C07322=1188.641,207.407,-59.713,-177.679,6.703,148.552
C07323=1188.636,207.656,-59.737,-177.676,6.705,148.552
C07324=1188.631,207.905,-59.762,-177.673,6.707,148.552
C07325=1188.627,208.154,-59.786,-177.671,6.709,148.551
C07326=1188.623,208.402,-59.810,-177.668,6.712,148.551
C07327=1188.618,208.651,-59.834,-177.665,6.713,148.551
C07328=1188.613,208.900,-59.858,-177.663,6.715,148.550
C07329=1188.609,209.149,-59.883,-177.660,6.717,148.550
C07330=1188.604,209.398,-59.907,-177.658,6.719,148.550
C07331=1188.599,209.646,-59.932,-177.654,6.722,148.550
C07332=1188.595,209.895,-59.956,-177.652,6.724,148.549
C07333=1188.591,210.144,-59.980,-177.650,6.726,148.549
C07334=1188.586,210.414,-60.007,-177.647,6.728,148.549
C07335=1188.581,210.684,-60.034,-177.644,6.730,148.549
C07336=1188.576,210.955,-60.061,-177.641,6.732,148.548
C07337=1188.571,211.226,-60.087,-177.638,6.735,148.548
C07338=1188.566,211.474,-60.111,-177.635,6.736,148.548
C07339=1188.561,211.722,-60.136,-177.633,6.738,148.547
C07340=1188.558,211.972,-60.161,-177.630,6.741,148.547
C07341=1188.552,212.220,-60.186,-177.627,6.743,148.547
C07342=1188.548,212.469,-60.210,-177.624,6.745,148.547
C07343=1188.543,212.718,-60.235,-177.622,6.747,148.546
C07344=1188.539,212.967,-60.259,-177.619,6.750,148.546
C07345=1188.534,213.215,-60.283,-177.616,6.751,148.546
C07346=1188.530,213.464,-60.308,-177.614,6.753,148.545
C07347=1188.525,213.713,-60.332,-177.612,6.755,148.545
C07348=1188.521,213.962,-60.358,-177.609,6.757,148.545
C07349=1188.516,214.210,-60.382,-177.606,6.760,148.545
C07350=1188.511,214.459,-60.407,-177.604,6.762,148.545
C07351=1188.507,214.708,-60.431,-177.601,6.764,148.544
C07352=1188.502,214.957,-60.456,-177.598,6.766,148.544
C07353=1188.498,215.205,-60.481,-177.595,6.768,148.544
C07354=1188.494,215.454,-60.506,-177.593,6.770,148.543
C07355=1188.489,215.703,-60.531,-177.590,6.772,148.543
C07356=1188.485,215.952,-60.555,-177.588,6.774,148.543
C07357=1188.480,216.200,-60.580,-177.585,6.777,148.543
C07358=1188.475,216.449,-60.605,-177.582,6.779,148.542
C07359=1188.471,216.698,-60.630,-177.580,6.781,148.542
C07360=1188.466,216.947,-60.654,-177.577,6.782,148.542
C07361=1188.462,217.195,-60.680,-177.574,6.785,148.542
C07362=1188.457,217.444,-60.704,-177.571,6.787,148.541
C07363=1188.453,217.693,-60.729,-177.569,6.789,148.541
C07364=1188.448,217.941,-60.754,-177.567,6.791,148.541
C07365=1188.444,218.190,-60.779,-177.563,6.794,148.541
C07366=1188.439,218.439,-60.804,-177.561,6.796,148.540
C07367=1188.434,218.687,-60.829,-177.559,6.798,148.540
C07368=1188.430,218.936,-60.853,-177.556,6.800,148.540
C07369=1188.426,219.185,-60.879,-177.553,6.802,148.539
C07370=1188.421,219.434,-60.904,-177.551,6.804,148.539
C07371=1188.417,219.682,-60.929,-177.548,6.806,148.539
C07372=1188.412,219.931,-60.954,-177.545,6.809,148.539
C07373=1188.407,220.180,-60.978,-177.543,6.811,148.539
C07374=1188.403,220.429,-61.004,-177.540,6.813,148.538
C07375=1188.399,220.677,-61.028,-177.537,6.815,148.538
C07376=1188.394,220.926,-61.054,-177.534,6.818,148.538
C07377=1188.389,221.175,-61.079,-177.532,6.819,148.538
C07378=1188.385,221.423,-61.104,-177.529,6.821,148.537
C07379=1188.380,221.672,-61.129,-177.527,6.823,148.537
C07380=1188.376,221.921,-61.154,-177.524,6.826,148.537
C07381=1188.371,222.169,-61.179,-177.521,6.828,148.536
C07382=1188.367,222.418,-61.205,-177.519,6.830,148.536
C07383=1188.362,222.666,-61.230,-177.516,6.833,148.536
C07384=1188.358,222.916,-61.255,-177.513,6.834,148.536
C07385=1188.353,223.164,-61.280,-177.511,6.837,148.536
C07386=1188.349,223.413,-61.305,-177.508,6.838,148.535
C07387=1188.345,223.662,-61.331,-177.506,6.841,148.535
C07388=1188.340,223.910,-61.356,-177.503,6.843,148.535
C07389=1188.336,224.159,-61.381,-177.500,6.845,148.535
C07390=1188.331,224.407,-61.406,-177.497,6.848,148.534
C07391=1188.327,224.656,-61.432,-177.495,6.850,148.534
C07392=1188.321,224.905,-61.457,-177.492,6.852,148.534
C07393=1188.317,225.154,-61.482,-177.489,6.855,148.534
C07394=1188.313,225.403,-61.508,-177.487,6.856,148.533
C07395=1188.309,225.651,-61.532,-177.485,6.859,148.533
C07396=1188.304,225.900,-61.558,-177.482,6.860,148.533
C07397=1188.300,226.148,-61.583,-177.479,6.863,148.533
C07398=1188.295,226.397,-61.609,-177.477,6.865,148.533
C07399=1188.291,226.646,-61.634,-177.474,6.867,148.532
C07400=1188.286,226.894,-61.660,-177.471,6.870,148.532
C07401=1188.282,227.143,-61.685,-177.469,6.872,148.532
C07402=1188.277,227.391,-61.711,-177.466,6.874,148.531
C07403=1188.273,227.640,-61.737,-177.463,6.877,148.531
C07404=1188.268,227.889,-61.762,-177.461,6.878,148.531
C07405=1188.263,228.137,-61.787,-177.458,6.880,148.531
C07406=1188.259,228.386,-61.813,-177.455,6.883,148.531
C07407=1188.255,228.635,-61.838,-177.452,6.885,148.530
C07408=1188.250,228.883,-61.864,-177.450,6.887,148.530
C07409=1188.246,229.132,-61.890,-177.447,6.890,148.530
C07410=1188.241,229.381,-61.915,-177.445,6.892,148.530
C07411=1188.236,229.629,-61.940,-177.442,6.894,148.529
C07412=1188.232,229.878,-61.966,-177.439,6.896,148.529
C07413=1188.228,230.127,-61.991,-177.437,6.899,148.529
C07414=1188.223,230.375,-62.017,-177.434,6.900,148.529
C07415=1188.218,230.624,-62.043,-177.432,6.903,148.529
C07416=1188.214,230.873,-62.069,-177.429,6.905,148.528
C07417=1188.209,231.121,-62.094,-177.427,6.907,148.528
C07418=1188.205,231.370,-62.120,-177.424,6.910,148.528
C07419=1188.201,231.619,-62.146,-177.421,6.912,148.528
C07420=1188.196,231.867,-62.171,-177.419,6.914,148.528
C07421=1188.192,232.116,-62.197,-177.415,6.917,148.527
C07422=1188.187,232.365,-62.223,-177.413,6.919,148.527
C07423=1188.183,232.613,-62.248,-177.411,6.921,148.527
C07424=1188.178,232.862,-62.274,-177.408,6.924,148.527
C07425=1188.173,233.111,-62.300,-177.405,6.925,148.526
C07426=1188.169,233.359,-62.326,-177.403,6.927,148.526
C07427=1188.165,233.608,-62.352,-177.400,6.930,148.526
C07428=1188.160,233.856,-62.378,-177.398,6.932,148.526
C07429=1188.155,234.105,-62.404,-177.395,6.934,148.526
C07430=1188.151,234.354,-62.430,-177.392,6.937,148.526
C07431=1188.147,234.602,-62.456,-177.390,6.939,148.525
C07432=1188.142,234.850,-62.481,-177.386,6.942,148.525
C07433=1188.138,235.099,-62.507,-177.384,6.944,148.525
C07434=1188.133,235.348,-62.533,-177.382,6.946,148.524
C07435=1188.129,235.597,-62.560,-177.379,6.949,148.524
C07436=1188.125,235.845,-62.585,-177.376,6.950,148.524
C07437=1188.120,236.093,-62.611,-177.374,6.952,148.524
C07438=1188.115,236.366,-62.639,-177.371,6.955,148.524
C07439=1188.110,236.637,-62.668,-177.368,6.958,148.524
C07440=1188.106,236.909,-62.696,-177.365,6.961,148.523
C07441=1188.101,237.179,-62.725,-177.362,6.963,148.523
C07442=1188.096,237.429,-62.751,-177.360,6.966,148.523
C07443=1188.091,237.677,-62.777,-177.357,6.967,148.523
C07444=1188.087,237.926,-62.803,-177.355,6.970,148.523
C07445=1188.082,238.175,-62.829,-177.352,6.972,148.522
C07446=1188.078,238.423,-62.855,-177.349,6.974,148.522
C07447=1188.074,238.671,-62.881,-177.346,6.977,148.522
C07448=1188.069,238.920,-62.908,-177.344,6.979,148.522
C07449=1188.065,239.169,-62.933,-177.341,6.981,148.521
C07450=1188.061,239.417,-62.960,-177.339,6.984,148.521
C07451=1188.056,239.666,-62.986,-177.336,6.986,148.521
C07452=1188.051,239.915,-63.012,-177.333,6.989,148.521
C07453=1188.047,240.162,-63.038,-177.331,6.991,148.521
C07454=1188.042,240.412,-63.064,-177.328,6.993,148.521
C07455=1188.038,240.660,-63.091,-177.326,6.996,148.521
C07456=1188.033,240.909,-63.117,-177.323,6.998,148.520
C07457=1188.029,241.157,-63.144,-177.320,7.001,148.520
C07458=1188.025,241.406,-63.169,-177.318,7.002,148.520
C07459=1188.020,241.654,-63.197,-177.316,7.004,148.520
C07460=1188.016,241.903,-63.222,-177.312,7.007,148.519
C07461=1188.011,242.152,-63.249,-177.310,7.009,148.519
C07462=1188.007,242.400,-63.275,-177.307,7.012,148.519
C07463=1188.002,242.648,-63.302,-177.305,7.014,148.519
C07464=1187.998,242.897,-63.328,-177.302,7.016,148.519
C07465=1187.993,243.146,-63.355,-177.299,7.019,148.519
C07466=1187.989,243.394,-63.380,-177.297,7.021,148.518
C07467=1187.984,243.643,-63.407,-177.294,7.024,148.518
C07468=1187.980,243.892,-63.433,-177.292,7.026,148.518
C07469=1187.975,244.140,-63.460,-177.289,7.029,148.518
C07470=1187.971,244.388,-63.487,-177.287,7.031,148.518
C07471=1187.966,244.637,-63.513,-177.284,7.033,148.517
C07472=1187.962,244.886,-63.540,-177.281,7.036,148.517
C07473=1187.958,245.134,-63.567,-177.279,7.038,148.517
C07474=1187.954,245.383,-63.592,-177.276,7.040,148.517
C07475=1187.949,245.631,-63.619,-177.274,7.042,148.517
C07476=1187.945,245.880,-63.646,-177.270,7.045,148.517
C07477=1187.940,246.129,-63.672,-177.268,7.047,148.516
C07478=1187.936,246.377,-63.699,-177.265,7.050,148.516
C07479=1187.931,246.625,-63.726,-177.263,7.052,148.516
C07480=1187.927,246.875,-63.752,-177.261,7.054,148.516
C07481=1187.923,247.123,-63.779,-177.258,7.057,148.516
C07482=1187.918,247.371,-63.806,-177.255,7.059,148.516
C07483=1187.914,247.619,-63.832,-177.252,7.062,148.515
C07484=1187.909,247.869,-63.858,-177.250,7.064,148.515
C07485=1187.904,248.117,-63.885,-177.247,7.067,148.515
C07486=1187.900,248.365,-63.912,-177.245,7.069,148.515
C07487=1187.896,248.614,-63.939,-177.242,7.072,148.515
C07488=1187.891,248.862,-63.966,-177.240,7.074,148.515
C07489=1187.887,249.110,-63.993,-177.237,7.076,148.514
C07490=1187.882,249.359,-64.019,-177.234,7.079,148.514
C07491=1187.878,249.608,-64.046,-177.232,7.080,148.514
C07492=1187.874,249.856,-64.072,-177.229,7.083,148.514
C07493=1187.869,250.105,-64.099,-177.227,7.086,148.514
C07494=1187.864,250.353,-64.127,-177.224,7.088,148.514
C07495=1187.860,250.602,-64.154,-177.221,7.090,148.514
C07496=1187.856,250.851,-64.180,-177.219,7.093,148.513
C07497=1187.852,251.099,-64.207,-177.216,7.095,148.513
C07498=1187.847,251.348,-64.235,-177.213,7.098,148.513
C07499=1187.842,251.596,-64.262,-177.211,7.100,148.513
C07500=1187.839,251.844,-64.288,-177.208,7.103,148.513
C07501=1187.834,252.093,-64.315,-177.206,7.105,148.513
C07502=1187.829,252.341,-64.342,-177.203,7.108,148.512
C07503=1187.825,252.590,-64.369,-177.200,7.110,148.512
C07504=1187.821,252.838,-64.396,-177.198,7.113,148.512
C07505=1187.817,253.087,-64.423,-177.195,7.115,148.512
C07506=1187.812,253.336,-64.450,-177.192,7.118,148.512
C07507=1187.807,253.584,-64.477,-177.190,7.120,148.512
C07508=1187.803,253.833,-64.504,-177.187,7.123,148.511
C07509=1187.799,254.081,-64.531,-177.185,7.125,148.511
C07510=1187.794,254.329,-64.558,-177.182,7.128,148.511
C07511=1187.789,254.578,-64.585,-177.180,7.130,148.511
C07512=1187.785,254.827,-64.612,-177.177,7.133,148.511
C07513=1187.781,255.075,-64.639,-177.175,7.135,148.511
C07514=1187.776,255.323,-64.667,-177.171,7.137,148.511
C07515=1187.772,255.572,-64.694,-177.169,7.140,148.510
C07516=1187.768,255.820,-64.721,-177.167,7.143,148.510
C07517=1187.764,256.069,-64.748,-177.164,7.145,148.510
C07518=1187.759,256.318,-64.775,-177.161,7.147,148.510
C07519=1187.755,256.566,-64.803,-177.159,7.150,148.510
C07520=1187.750,256.814,-64.830,-177.156,7.153,148.510
C07521=1187.745,257.063,-64.857,-177.154,7.154,148.510
C07522=1187.741,257.312,-64.885,-177.151,7.157,148.510
C07523=1187.737,257.560,-64.912,-177.149,7.160,148.509
C07524=1187.732,257.808,-64.939,-177.146,7.162,148.509
C07525=1187.728,258.057,-64.966,-177.143,7.165,148.509
C07526=1187.723,258.305,-64.993,-177.141,7.167,148.509
C07527=1187.719,258.554,-65.022,-177.138,7.170,148.509
C07528=1187.715,258.802,-65.049,-177.135,7.172,148.509
C07529=1187.710,259.051,-65.076,-177.133,7.175,148.509
C07530=1187.706,259.299,-65.104,-177.130,7.177,148.509
C07531=1187.702,259.548,-65.131,-177.127,7.180,148.508
C07532=1187.697,259.796,-65.158,-177.125,7.182,148.508
C07533=1187.693,260.044,-65.186,-177.122,7.185,148.508
C07534=1187.688,260.293,-65.213,-177.120,7.187,148.508
C07535=1187.684,260.541,-65.241,-177.117,7.190,148.508
C07536=1187.679,260.790,-65.268,-177.115,7.192,148.508
C07537=1187.675,261.038,-65.295,-177.112,7.195,148.508
C07538=1187.671,261.287,-65.323,-177.109,7.198,148.508
C07539=1187.666,261.535,-65.350,-177.107,7.200,148.507
C07540=1187.662,261.783,-65.378,-177.104,7.203,148.507
C07541=1187.657,262.032,-65.405,-177.102,7.205,148.507
C07542=1187.653,262.305,-65.436,-177.099,7.208,148.507
C07543=1187.647,262.578,-65.466,-177.096,7.211,148.507
C07544=1187.644,262.851,-65.496,-177.093,7.214,148.507
C07545=1187.638,263.123,-65.527,-177.090,7.216,148.507
C07546=1187.635,263.372,-65.555,-177.088,7.219,148.506
C07547=1187.630,263.620,-65.582,-177.085,7.222,148.506
C07548=1187.625,263.868,-65.610,-177.082,7.224,148.506
C07549=1187.621,264.118,-65.638,-177.080,7.226,148.506
C07550=1187.616,264.366,-65.665,-177.077,7.229,148.506
C07551=1187.612,264.613,-65.693,-177.075,7.231,148.506
C07552=1187.608,264.863,-65.721,-177.072,7.234,148.506
C07553=1187.603,265.111,-65.749,-177.070,7.236,148.506
C07554=1187.598,265.359,-65.776,-177.067,7.239,148.506
C07555=1187.594,265.608,-65.804,-177.064,7.242,148.505
C07556=1187.590,265.856,-65.832,-177.062,7.244,148.505
C07557=1187.586,266.105,-65.859,-177.059,7.247,148.505
C07558=1187.581,266.353,-65.888,-177.057,7.249,148.505
C07559=1187.577,266.601,-65.915,-177.054,7.252,148.505
C07560=1187.573,266.850,-65.944,-177.051,7.255,148.505
C07561=1187.568,267.098,-65.971,-177.049,7.257,148.505
C07562=1187.564,267.347,-65.999,-177.046,7.260,148.505
C07563=1187.559,267.595,-66.027,-177.044,7.262,148.505
C07564=1187.555,267.843,-66.055,-177.041,7.265,148.504
C07565=1187.551,268.092,-66.082,-177.038,7.268,148.504
C07566=1187.546,268.340,-66.111,-177.036,7.270,148.504
C07567=1187.542,268.589,-66.139,-177.033,7.273,148.504
C07568=1187.538,268.837,-66.167,-177.031,7.275,148.504
C07569=1187.533,269.085,-66.195,-177.028,7.278,148.504
C07570=1187.529,269.334,-66.222,-177.025,7.281,148.504
C07571=1187.524,269.582,-66.250,-177.023,7.283,148.504
C07572=1187.520,269.831,-66.279,-177.020,7.286,148.504
C07573=1187.515,270.079,-66.307,-177.018,7.289,148.504
C07574=1187.512,270.327,-66.335,-177.015,7.291,148.503
C07575=1187.507,270.575,-66.363,-177.012,7.294,148.503
C07576=1187.503,270.824,-66.391,-177.010,7.296,148.503
C07577=1187.498,271.072,-66.420,-177.007,7.299,148.503
C07578=1187.494,271.321,-66.448,-177.005,7.302,148.503
C07579=1187.490,271.569,-66.476,-177.002,7.304,148.503
C07580=1187.485,271.817,-66.504,-176.999,7.307,148.503
C07581=1187.481,272.065,-66.532,-176.997,7.309,148.503
C07582=1187.476,272.314,-66.561,-176.994,7.312,148.503
C07583=1187.472,272.562,-66.589,-176.992,7.315,148.503
C07584=1187.468,272.811,-66.617,-176.990,7.317,148.503
C07585=1187.463,273.059,-66.645,-176.987,7.320,148.503
C07586=1187.459,273.307,-66.673,-176.984,7.323,148.502
C07587=1187.454,273.556,-66.702,-176.981,7.325,148.502
C07588=1187.451,273.804,-66.730,-176.979,7.328,148.502
C07589=1187.445,274.052,-66.758,-176.977,7.330,148.502
C07590=1187.442,274.301,-66.786,-176.974,7.333,148.502
C07591=1187.437,274.550,-66.815,-176.971,7.336,148.502
C07592=1187.433,274.798,-66.843,-176.969,7.339,148.502
C07593=1187.428,275.047,-66.872,-176.966,7.342,148.502
C07594=1187.424,275.294,-66.899,-176.963,7.344,148.502
C07595=1187.420,275.543,-66.929,-176.961,7.346,148.502
C07596=1187.416,275.791,-66.957,-176.958,7.349,148.502
C07597=1187.411,276.040,-66.985,-176.955,7.352,148.502
C07598=1187.407,276.288,-67.014,-176.953,7.355,148.501
C07599=1187.402,276.536,-67.042,-176.951,7.358,148.501
C07600=1187.399,276.784,-67.071,-176.948,7.361,148.501
C07601=1187.394,277.032,-67.099,-176.946,7.363,148.501
C07602=1187.389,277.281,-67.128,-176.943,7.366,148.501
C07603=1187.385,277.530,-67.156,-176.940,7.368,148.501
C07604=1187.381,277.777,-67.185,-176.938,7.371,148.501
C07605=1187.377,278.026,-67.213,-176.935,7.374,148.501
C07606=1187.372,278.274,-67.242,-176.932,7.377,148.501
C07607=1187.368,278.522,-67.271,-176.930,7.379,148.501
C07608=1187.364,278.771,-67.299,-176.927,7.382,148.501
C07609=1187.359,279.019,-67.328,-176.925,7.385,148.501
C07610=1187.355,279.268,-67.357,-176.922,7.387,148.501
C07611=1187.351,279.516,-67.385,-176.920,7.390,148.501
C07612=1187.346,279.764,-67.414,-176.917,7.393,148.501
C07613=1187.342,280.013,-67.443,-176.915,7.395,148.500
C07614=1187.338,280.261,-67.471,-176.912,7.398,148.500
C07615=1187.333,280.509,-67.500,-176.909,7.401,148.500
C07616=1187.329,280.758,-67.529,-176.907,7.403,148.500
C07617=1187.325,281.006,-67.557,-176.904,7.406,148.500
C07618=1187.320,281.254,-67.586,-176.901,7.409,148.500
C07619=1187.316,281.503,-67.615,-176.899,7.411,148.500
C07620=1187.312,281.751,-67.644,-176.896,7.414,148.500
C07621=1187.308,281.999,-67.673,-176.894,7.417,148.500
C07622=1187.303,282.247,-67.702,-176.892,7.419,148.500
C07623=1187.298,282.496,-67.730,-176.889,7.422,148.500
C07624=1187.294,282.744,-67.760,-176.886,7.425,148.500
C07625=1187.290,282.992,-67.788,-176.884,7.427,148.500
C07626=1187.286,283.240,-67.817,-176.881,7.430,148.500
C07627=1187.281,283.489,-67.846,-176.879,7.433,148.500
C07628=1187.277,283.737,-67.875,-176.876,7.436,148.500
C07629=1187.272,283.986,-67.904,-176.874,7.438,148.499
C07630=1187.268,284.234,-67.933,-176.871,7.441,148.499
C07631=1187.264,284.482,-67.962,-176.868,7.444,148.499
C07632=1187.260,284.731,-67.991,-176.866,7.447,148.499
C07633=1187.255,284.978,-68.020,-176.863,7.450,148.499
C07634=1187.251,285.227,-68.049,-176.860,7.452,148.499
C07635=1187.246,285.475,-68.078,-176.858,7.454,148.499
C07636=1187.243,285.723,-68.107,-176.855,7.457,148.499
C07637=1187.238,285.971,-68.136,-176.853,7.460,148.499
C07638=1187.234,286.220,-68.165,-176.850,7.463,148.499
C07639=1187.229,286.468,-68.194,-176.848,7.466,148.499
C07640=1187.225,286.716,-68.224,-176.845,7.469,148.499
C07641=1187.221,286.965,-68.253,-176.842,7.472,148.499
C07642=1187.216,287.213,-68.281,-176.840,7.475,148.499
C07643=1187.212,287.461,-68.311,-176.837,7.477,148.499
C07644=1187.208,287.709,-68.340,-176.835,7.480,148.499
C07645=1187.203,287.958,-68.370,-176.832,7.483,148.499
C07646=1187.199,288.232,-68.401,-176.829,7.486,148.499
C07647=1187.194,288.507,-68.433,-176.827,7.489,148.499
C07648=1187.189,288.781,-68.466,-176.824,7.492,148.499
C07649=1187.185,289.056,-68.498,-176.821,7.495,148.498
C07650=1187.180,289.304,-68.527,-176.818,7.498,148.498
C07651=1187.176,289.552,-68.557,-176.816,7.501,148.498
C07652=1187.172,289.800,-68.586,-176.814,7.503,148.498
C07653=1187.168,290.049,-68.616,-176.811,7.506,148.498
C07654=1187.163,290.297,-68.645,-176.808,7.509,148.498
C07655=1187.159,290.546,-68.674,-176.805,7.512,148.498
C07656=1187.155,290.794,-68.703,-176.803,7.514,148.498
C07657=1187.150,291.042,-68.733,-176.801,7.517,148.498
C07658=1187.145,291.290,-68.763,-176.798,7.520,148.498
C07659=1187.141,291.538,-68.792,-176.795,7.523,148.498
C07660=1187.137,291.787,-68.822,-176.793,7.525,148.498
C07661=1187.133,292.035,-68.851,-176.790,7.528,148.498
C07662=1187.128,292.283,-68.880,-176.787,7.531,148.498
C07663=1187.124,292.532,-68.910,-176.785,7.534,148.498
C07664=1187.120,292.780,-68.939,-176.783,7.536,148.498
C07665=1187.116,293.028,-68.969,-176.780,7.540,148.498
C07666=1187.112,293.276,-68.999,-176.778,7.543,148.498
C07667=1187.108,293.524,-69.028,-176.775,7.546,148.498
C07668=1187.104,293.772,-69.058,-176.773,7.548,148.498
C07669=1187.099,294.021,-69.088,-176.770,7.551,148.498
C07670=1187.094,294.268,-69.117,-176.767,7.554,148.498
C07671=1187.090,294.517,-69.146,-176.765,7.557,148.498
C07672=1187.086,294.765,-69.176,-176.762,7.559,148.498
C07673=1187.081,295.013,-69.205,-176.760,7.562,148.498
C07674=1187.077,295.261,-69.235,-176.757,7.565,148.498
C07675=1187.073,295.509,-69.266,-176.754,7.568,148.498
C07676=1187.068,295.758,-69.295,-176.752,7.570,148.498
C07677=1187.064,296.006,-69.324,-176.749,7.573,148.498
C07678=1187.060,296.254,-69.354,-176.747,7.576,148.498
C07679=1187.056,296.502,-69.384,-176.745,7.580,148.498
C07680=1187.051,296.750,-69.414,-176.742,7.582,148.498
C07681=1187.047,296.999,-69.444,-176.740,7.585,148.498
C07682=1187.043,297.247,-69.473,-176.737,7.588,148.498
C07683=1187.039,297.495,-69.503,-176.734,7.591,148.498
C07684=1187.034,297.743,-69.533,-176.731,7.594,148.498
C07685=1187.030,297.991,-69.563,-176.729,7.596,148.498
C07686=1187.026,298.239,-69.593,-176.727,7.599,148.498
C07687=1187.022,298.487,-69.622,-176.724,7.602,148.498
C07688=1187.017,298.736,-69.652,-176.721,7.605,148.498
C07689=1187.013,298.984,-69.683,-176.720,7.607,148.498
C07690=1187.009,299.233,-69.712,-176.717,7.610,148.498
C07691=1187.004,299.481,-69.742,-176.714,7.613,148.498
C07692=1187.001,299.729,-69.773,-176.711,7.616,148.498
C07693=1186.996,299.977,-69.802,-176.709,7.619,148.498
C07694=1186.992,300.225,-69.833,-176.706,7.622,148.498
C07695=1186.988,300.473,-69.862,-176.704,7.625,148.497
C07696=1186.983,300.722,-69.892,-176.702,7.628,148.498
C07697=1186.979,300.970,-69.922,-176.699,7.631,148.498
C07698=1186.975,301.218,-69.952,-176.696,7.634,148.498
C07699=1186.971,301.465,-69.982,-176.694,7.636,148.498
C07700=1186.966,301.714,-70.012,-176.691,7.639,148.498
C07701=1186.962,301.962,-70.042,-176.689,7.642,148.498
C07702=1186.958,302.211,-70.073,-176.686,7.645,148.498
C07703=1186.954,302.459,-70.103,-176.684,7.648,148.498
C07704=1186.949,302.707,-70.133,-176.681,7.651,148.498
C07705=1186.945,302.955,-70.163,-176.679,7.654,148.498
C07706=1186.941,303.202,-70.193,-176.676,7.657,148.498
C07707=1186.936,303.451,-70.223,-176.673,7.660,148.498
C07708=1186.932,303.699,-70.254,-176.671,7.663,148.498
C07709=1186.927,303.947,-70.284,-176.669,7.665,148.498
C07710=1186.924,304.195,-70.314,-176.666,7.668,148.498
C07711=1186.920,304.444,-70.345,-176.663,7.671,148.498
C07712=1186.915,304.692,-70.374,-176.661,7.674,148.498
C07713=1186.911,304.940,-70.405,-176.658,7.677,148.498
C07714=1186.907,305.187,-70.435,-176.656,7.680,148.498
C07715=1186.902,305.436,-70.465,-176.654,7.683,148.498
C07716=1186.898,305.684,-70.495,-176.651,7.686,148.498
C07717=1186.894,305.932,-70.527,-176.648,7.689,148.498
C07718=1186.889,306.181,-70.557,-176.645,7.692,148.498
C07719=1186.885,306.429,-70.587,-176.643,7.695,148.498
C07720=1186.881,306.676,-70.618,-176.641,7.697,148.498
C07721=1186.877,306.924,-70.648,-176.638,7.700,148.498
C07722=1186.873,307.173,-70.679,-176.636,7.703,148.498
C07723=1186.869,307.421,-70.708,-176.633,7.706,148.498
C07724=1186.864,307.669,-70.739,-176.631,7.709,148.498
C07725=1186.859,307.917,-70.770,-176.629,7.712,148.498
C07726=1186.855,308.165,-70.800,-176.626,7.715,148.498
C07727=1186.851,308.413,-70.831,-176.623,7.718,148.498
C07728=1186.847,308.661,-70.862,-176.621,7.721,148.498
C07729=1186.843,308.910,-70.891,-176.618,7.724,148.498
C07730=1186.838,309.157,-70.922,-176.615,7.727,148.498
C07731=1186.835,309.406,-70.953,-176.613,7.729,148.498
C07732=1186.830,309.654,-70.983,-176.611,7.732,148.498
C07733=1186.826,309.902,-71.014,-176.608,7.735,148.498
C07734=1186.822,310.149,-71.044,-176.606,7.738,148.498
C07735=1186.818,310.398,-71.075,-176.603,7.741,148.498
C07736=1186.813,310.646,-71.106,-176.601,7.745,148.498
C07737=1186.808,310.894,-71.137,-176.599,7.747,148.498
C07738=1186.805,311.142,-71.168,-176.596,7.750,148.498
C07739=1186.801,311.390,-71.198,-176.593,7.753,148.498
C07740=1186.796,311.638,-71.229,-176.591,7.756,148.498
C07741=1186.792,311.886,-71.259,-176.588,7.759,148.498
C07742=1186.788,312.135,-71.290,-176.585,7.762,148.498
C07743=1186.783,312.382,-71.321,-176.584,7.765,148.499
C07744=1186.779,312.630,-71.352,-176.581,7.768,148.499
C07745=1186.776,312.879,-71.382,-176.578,7.771,148.499
C07746=1186.771,313.127,-71.413,-176.576,7.774,148.499
C07747=1186.766,313.375,-71.444,-176.573,7.777,148.499
C07748=1186.762,313.623,-71.475,-176.571,7.780,148.499
C07749=1186.758,313.871,-71.507,-176.568,7.783,148.499
C07750=1186.754,314.148,-71.541,-176.566,7.786,148.499
C07751=1186.749,314.424,-71.575,-176.563,7.789,148.499
C07752=1186.744,314.700,-71.610,-176.560,7.792,148.499
C07753=1186.739,314.978,-71.644,-176.557,7.796,148.499
C07754=1186.735,315.226,-71.675,-176.555,7.800,148.499
C07755=1186.730,315.473,-71.706,-176.553,7.802,148.499
C07756=1186.727,315.721,-71.737,-176.550,7.805,148.499
C07757=1186.723,315.969,-71.767,-176.548,7.808,148.499
C07758=1186.719,316.218,-71.799,-176.545,7.811,148.499
C07759=1186.714,316.465,-71.830,-176.542,7.814,148.499
C07760=1186.710,316.713,-71.861,-176.540,7.817,148.500
C07761=1186.706,316.962,-71.892,-176.537,7.820,148.499
C07762=1186.701,317.209,-71.923,-176.535,7.823,148.499
C07763=1186.697,317.458,-71.955,-176.533,7.826,148.500
C07764=1186.693,317.706,-71.985,-176.530,7.829,148.500
C07765=1186.689,317.953,-72.016,-176.527,7.832,148.500
C07766=1186.685,318.201,-72.047,-176.525,7.835,148.500
C07767=1186.680,318.449,-72.078,-176.522,7.838,148.500
C07768=1186.677,318.697,-72.110,-176.520,7.841,148.500
C07769=1186.672,318.945,-72.141,-176.518,7.844,148.500
C07770=1186.668,319.193,-72.173,-176.515,7.847,148.500
C07771=1186.664,319.441,-72.203,-176.513,7.850,148.500
C07772=1186.660,319.690,-72.235,-176.510,7.853,148.500
C07773=1186.655,319.937,-72.266,-176.508,7.856,148.500
C07774=1186.651,320.185,-72.297,-176.505,7.859,148.500
C07775=1186.647,320.433,-72.329,-176.503,7.862,148.500
C07776=1186.643,320.681,-72.359,-176.500,7.866,148.501
C07777=1186.639,320.929,-72.391,-176.498,7.868,148.500
C07778=1186.634,321.177,-72.422,-176.496,7.871,148.501
C07779=1186.631,321.425,-72.454,-176.493,7.874,148.501
C07780=1186.626,321.673,-72.485,-176.491,7.877,148.501
C07781=1186.622,321.921,-72.516,-176.488,7.880,148.501
C07782=1186.617,322.170,-72.548,-176.486,7.883,148.501
C07783=1186.613,322.418,-72.580,-176.483,7.887,148.501
C07784=1186.609,322.666,-72.611,-176.481,7.890,148.501
C07785=1186.605,322.914,-72.642,-176.479,7.892,148.501
C07786=1186.601,323.162,-72.674,-176.476,7.895,148.501
C07787=1186.597,323.409,-72.706,-176.474,7.899,148.501
C07788=1186.593,323.658,-72.737,-176.471,7.902,148.501
C07789=1186.589,323.905,-72.768,-176.469,7.905,148.502
C07790=1186.585,324.153,-72.800,-176.466,7.908,148.502
C07791=1186.580,324.401,-72.831,-176.464,7.911,148.502
C07792=1186.576,324.649,-72.863,-176.461,7.914,148.502
C07793=1186.571,324.897,-72.895,-176.459,7.918,148.502
C07794=1186.567,325.145,-72.926,-176.457,7.920,148.502
C07795=1186.564,325.393,-72.958,-176.455,7.923,148.502
C07796=1186.559,325.641,-72.989,-176.452,7.926,148.502
C07797=1186.556,325.889,-73.021,-176.450,7.929,148.502
C07798=1186.550,326.137,-73.052,-176.447,7.932,148.502
C07799=1186.547,326.385,-73.084,-176.445,7.936,148.503
C07800=1186.543,326.633,-73.116,-176.442,7.939,148.503
C07801=1186.539,326.880,-73.148,-176.440,7.942,148.503
C07802=1186.534,327.129,-73.180,-176.437,7.945,148.503
C07803=1186.530,327.377,-73.211,-176.436,7.948,148.503
C07804=1186.526,327.625,-73.243,-176.433,7.951,148.503
C07805=1186.522,327.873,-73.274,-176.431,7.954,148.503
C07806=1186.517,328.121,-73.306,-176.428,7.957,148.503
C07807=1186.513,328.369,-73.338,-176.426,7.960,148.503
C07808=1186.510,328.617,-73.370,-176.423,7.963,148.503
C07809=1186.505,328.864,-73.402,-176.421,7.967,148.504
C07810=1186.501,329.112,-73.434,-176.418,7.970,148.504
C07811=1186.497,329.360,-73.466,-176.416,7.973,148.504
C07812=1186.493,329.608,-73.497,-176.413,7.976,148.504
C07813=1186.488,329.856,-73.530,-176.411,7.978,148.504
C07814=1186.484,330.103,-73.561,-176.409,7.982,148.504
C07815=1186.480,330.352,-73.592,-176.407,7.985,148.504
C07816=1186.476,330.600,-73.626,-176.404,7.988,148.504
C07817=1186.472,330.847,-73.657,-176.402,7.991,148.505
C07818=1186.467,331.095,-73.690,-176.399,7.994,148.505
C07819=1186.464,331.343,-73.721,-176.397,7.998,148.505
C07820=1186.460,331.591,-73.753,-176.395,8.001,148.505
C07821=1186.455,331.839,-73.785,-176.392,8.004,148.505
C07822=1186.451,332.087,-73.817,-176.390,8.007,148.505
C07823=1186.447,332.336,-73.850,-176.387,8.011,148.505
C07824=1186.442,332.583,-73.881,-176.385,8.013,148.505
C07825=1186.439,332.831,-73.913,-176.383,8.016,148.506
C07826=1186.434,333.079,-73.945,-176.380,8.019,148.506
C07827=1186.431,333.327,-73.977,-176.378,8.022,148.506
C07828=1186.426,333.574,-74.010,-176.376,8.026,148.506
C07829=1186.422,333.822,-74.042,-176.373,8.029,148.506
C07830=1186.418,334.071,-74.074,-176.371,8.032,148.506
C07831=1186.414,334.319,-74.106,-176.369,8.035,148.506
C07832=1186.409,334.566,-74.138,-176.366,8.039,148.507
C07833=1186.405,334.814,-74.171,-176.364,8.042,148.507
C07834=1186.401,335.062,-74.203,-176.361,8.045,148.507
C07835=1186.397,335.310,-74.235,-176.359,8.048,148.507
C07836=1186.392,335.558,-74.267,-176.357,8.051,148.507
C07837=1186.389,335.805,-74.300,-176.355,8.054,148.507
C07838=1186.384,336.054,-74.332,-176.352,8.057,148.507
C07839=1186.381,336.302,-74.364,-176.350,8.061,148.508
C07840=1186.376,336.549,-74.397,-176.348,8.064,148.508
C07841=1186.372,336.797,-74.429,-176.345,8.067,148.508
C07842=1186.368,337.045,-74.461,-176.343,8.070,148.508
C07843=1186.364,337.292,-74.494,-176.341,8.074,148.508
C07844=1186.360,337.541,-74.526,-176.338,8.077,148.508
C07845=1186.356,337.789,-74.558,-176.336,8.080,148.509
C07846=1186.352,338.036,-74.591,-176.334,8.083,148.509
C07847=1186.347,338.284,-74.623,-176.331,8.086,148.509
C07848=1186.344,338.532,-74.656,-176.329,8.089,148.509
C07849=1186.339,338.780,-74.688,-176.327,8.092,148.509
C07850=1186.335,339.028,-74.721,-176.325,8.095,148.509
C07851=1186.331,339.276,-74.753,-176.322,8.099,148.510
C07852=1186.326,339.523,-74.785,-176.320,8.102,148.510
C07853=1186.322,339.771,-74.818,-176.318,8.105,148.510
C07854=1186.318,340.050,-74.855,-176.315,8.109,148.510
C07855=1186.313,340.329,-74.891,-176.312,8.112,148.510
C07856=1186.309,340.608,-74.928,-176.310,8.116,148.511
C07857=1186.304,340.887,-74.965,-176.307,8.120,148.511
C07858=1186.301,341.134,-74.997,-176.305,8.123,148.511
C07859=1186.296,341.382,-75.030,-176.303,8.127,148.511
C07860=1186.291,341.630,-75.063,-176.300,8.130,148.511
C07861=1186.287,341.878,-75.095,-176.298,8.133,148.511
C07862=1186.284,342.126,-75.128,-176.296,8.135,148.512
C07863=1186.279,342.373,-75.161,-176.294,8.139,148.512
C07864=1186.275,342.622,-75.193,-176.292,8.142,148.512
C07865=1186.271,342.869,-75.226,-176.289,8.145,148.512
C07866=1186.267,343.117,-75.259,-176.287,8.149,148.512
C07867=1186.263,343.365,-75.291,-176.285,8.152,148.513
C07868=1186.259,343.613,-75.325,-176.283,8.155,148.513
C07869=1186.254,343.860,-75.357,-176.280,8.159,148.513
C07870=1186.250,344.108,-75.390,-176.278,8.162,148.513
C07871=1186.246,344.356,-75.422,-176.276,8.165,148.514
C07872=1186.242,344.603,-75.456,-176.273,8.168,148.514
C07873=1186.238,344.852,-75.488,-176.271,8.172,148.514
C07874=1186.234,345.100,-75.521,-176.269,8.175,148.514
C07875=1186.229,345.347,-75.554,-176.266,8.178,148.514
C07876=1186.225,345.595,-75.587,-176.264,8.182,148.514
C07877=1186.221,345.843,-75.621,-176.262,8.185,148.515
C07878=1186.217,346.091,-75.652,-176.260,8.188,148.515
C07879=1186.213,346.338,-75.686,-176.258,8.191,148.515
C07880=1186.209,346.586,-75.719,-176.256,8.194,148.515
C07881=1186.205,346.834,-75.752,-176.254,8.197,148.516
C07882=1186.201,347.082,-75.785,-176.252,8.201,148.516
C07883=1186.197,347.329,-75.818,-176.249,8.204,148.516
C07884=1186.192,347.578,-75.851,-176.247,8.208,148.516
C07885=1186.188,347.825,-75.884,-176.245,8.211,148.517
C07886=1186.184,348.073,-75.917,-176.243,8.214,148.517
C07887=1186.180,348.321,-75.950,-176.240,8.217,148.517
C07888=1186.176,348.569,-75.983,-176.238,8.221,148.517
C07889=1186.172,348.816,-76.016,-176.236,8.224,148.517
C07890=1186.168,349.064,-76.049,-176.234,8.227,148.518
C07891=1186.164,349.312,-76.082,-176.231,8.231,148.518
C07892=1186.160,349.559,-76.115,-176.229,8.234,148.518
C07893=1186.156,349.807,-76.148,-176.227,8.237,148.518
C07894=1186.152,350.055,-76.182,-176.225,8.241,148.519
C07895=1186.147,350.302,-76.215,-176.223,8.244,148.519
C07896=1186.143,350.550,-76.248,-176.221,8.248,148.519
C07897=1186.140,350.799,-76.281,-176.218,8.251,148.519
C07898=1186.136,351.046,-76.315,-176.216,8.254,148.520
C07899=1186.132,351.294,-76.348,-176.214,8.257,148.520
C07900=1186.127,351.542,-76.382,-176.213,8.260,148.520
C07901=1186.123,351.790,-76.415,-176.210,8.264,148.520
C07902=1186.119,352.037,-76.449,-176.208,8.267,148.521
C07903=1186.115,352.285,-76.482,-176.206,8.270,148.521
C07904=1186.110,352.532,-76.515,-176.204,8.274,148.521
C07905=1186.106,352.780,-76.548,-176.202,8.277,148.522
C07906=1186.102,353.028,-76.581,-176.200,8.281,148.522
C07907=1186.098,353.276,-76.614,-176.197,8.284,148.522
C07908=1186.095,353.523,-76.649,-176.195,8.287,148.522
C07909=1186.091,353.771,-76.682,-176.193,8.291,148.523
C07910=1186.086,354.019,-76.715,-176.191,8.294,148.523
C07911=1186.082,354.267,-76.748,-176.189,8.298,148.523
C07912=1186.077,354.515,-76.782,-176.187,8.301,148.524
C07913=1186.074,354.762,-76.816,-176.185,8.305,148.524
C07914=1186.070,355.009,-76.849,-176.182,8.308,148.524
C07915=1186.066,355.258,-76.882,-176.181,8.311,148.524
C07916=1186.062,355.505,-76.916,-176.178,8.315,148.525
C07917=1186.058,355.753,-76.949,-176.176,8.318,148.525
C07918=1186.053,356.001,-76.983,-176.174,8.322,148.525
C07919=1186.049,356.249,-77.016,-176.172,8.325,148.526
C07920=1186.045,356.496,-77.050,-176.170,8.328,148.526
C07921=1186.042,356.744,-77.084,-176.168,8.332,148.526
C07922=1186.038,356.991,-77.118,-176.166,8.335,148.526
C07923=1186.033,357.239,-77.151,-176.164,8.339,148.527
C07924=1186.029,357.487,-77.184,-176.162,8.342,148.527
C07925=1186.025,357.734,-77.218,-176.160,8.345,148.527
C07926=1186.021,357.982,-77.252,-176.158,8.348,148.528
C07927=1186.018,358.230,-77.286,-176.156,8.352,148.528
C07928=1186.013,358.478,-77.319,-176.154,8.355,148.528
C07929=1186.009,358.725,-77.353,-176.152,8.359,148.529
C07930=1186.005,358.973,-77.387,-176.150,8.362,148.529
C07931=1186.001,359.221,-77.420,-176.148,8.366,148.529
C07932=1185.997,359.468,-77.454,-176.146,8.369,148.530
C07933=1185.992,359.716,-77.488,-176.144,8.373,148.530
C07934=1185.989,359.963,-77.521,-176.142,8.376,148.530
C07935=1185.984,360.212,-77.556,-176.140,8.380,148.531
C07936=1185.981,360.459,-77.589,-176.138,8.383,148.531
C07937=1185.977,360.706,-77.623,-176.136,8.387,148.531
C07938=1185.972,360.955,-77.657,-176.134,8.390,148.532
C07939=1185.969,361.202,-77.691,-176.132,8.394,148.532
C07940=1185.964,361.450,-77.724,-176.131,8.396,148.532
C07941=1185.960,361.697,-77.759,-176.129,8.400,148.533
C07942=1185.957,361.945,-77.793,-176.127,8.403,148.533
C07943=1185.953,362.193,-77.826,-176.125,8.407,148.534
C07944=1185.948,362.440,-77.861,-176.123,8.410,148.534
C07945=1185.944,362.688,-77.894,-176.121,8.414,148.534
C07946=1185.941,362.936,-77.928,-176.119,8.418,148.535
C07947=1185.936,363.183,-77.963,-176.117,8.421,148.535
C07948=1185.932,363.431,-77.996,-176.116,8.424,148.535
C07949=1185.928,363.679,-78.031,-176.114,8.427,148.536
C07950=1185.924,363.926,-78.065,-176.112,8.431,148.536
C07951=1185.920,364.173,-78.098,-176.110,8.435,148.537
C07952=1185.916,364.422,-78.133,-176.108,8.438,148.537
C07953=1185.912,364.669,-78.166,-176.107,8.441,148.537
C07954=1185.908,364.916,-78.201,-176.105,8.444,148.538
C07955=1185.904,365.164,-78.235,-176.103,8.448,148.538
C07956=1185.899,365.412,-78.269,-176.101,8.452,148.538
C07957=1185.896,365.660,-78.303,-176.099,8.455,148.539
C07958=1185.891,365.941,-78.342,-176.098,8.459,148.539
C07959=1185.887,366.222,-78.381,-176.096,8.462,148.540
C07960=1185.882,366.504,-78.420,-176.093,8.467,148.540
C07961=1185.878,366.785,-78.459,-176.092,8.471,148.541
C07962=1185.873,367.033,-78.493,-176.090,8.474,148.541
C07963=1185.870,367.280,-78.526,-176.089,8.477,148.542
C07964=1185.866,367.528,-78.561,-176.087,8.481,148.542
C07965=1185.862,367.775,-78.595,-176.085,8.484,148.543
C07966=1185.857,368.023,-78.630,-176.084,8.488,148.543
C07967=1185.853,368.271,-78.664,-176.082,8.491,148.543
C07968=1185.849,368.518,-78.698,-176.080,8.495,148.544
C07969=1185.845,368.766,-78.733,-176.079,8.498,148.544
C07970=1185.842,369.013,-78.767,-176.077,8.501,148.545
C07971=1185.837,369.261,-78.801,-176.076,8.505,148.545
C07972=1185.834,369.508,-78.836,-176.074,8.508,148.545
C07973=1185.829,369.756,-78.869,-176.073,8.511,148.546
C07974=1185.825,370.005,-78.904,-176.071,8.515,148.547
C07975=1185.821,370.252,-78.938,-176.069,8.519,148.547
C07976=1185.817,370.500,-78.973,-176.068,8.521,148.547
C07977=1185.814,370.746,-79.008,-176.067,8.525,148.548
C07978=1185.809,370.994,-79.042,-176.065,8.529,148.548
C07979=1185.805,371.242,-79.077,-176.064,8.532,148.549
C07980=1185.801,371.489,-79.111,-176.062,8.535,148.549
C07981=1185.797,371.737,-79.146,-176.061,8.538,148.550
C07982=1185.793,371.984,-79.180,-176.059,8.542,148.550
C07983=1185.790,372.232,-79.214,-176.057,8.546,148.551
C07984=1185.785,372.480,-79.249,-176.057,8.549,148.551
C07985=1185.781,372.728,-79.284,-176.055,8.552,148.552
C07986=1185.777,372.975,-79.317,-176.054,8.555,148.552
C07987=1185.773,373.222,-79.352,-176.052,8.559,148.553
C07988=1185.769,373.470,-79.387,-176.051,8.562,148.553
C07989=1185.765,373.717,-79.421,-176.050,8.566,148.554
C07990=1185.761,373.965,-79.456,-176.048,8.569,148.554
C07991=1185.757,374.212,-79.491,-176.047,8.573,148.555
C07992=1185.753,374.460,-79.525,-176.046,8.575,148.555
C07993=1185.749,374.708,-79.559,-176.044,8.579,148.556
C07994=1185.745,374.955,-79.595,-176.043,8.582,148.556
C07995=1185.741,375.203,-79.629,-176.042,8.586,148.557
C07996=1185.737,375.450,-79.664,-176.041,8.589,148.557
C07997=1185.733,375.698,-79.698,-176.039,8.593,148.558
C07998=1185.729,375.946,-79.733,-176.038,8.595,148.558
C07999=1185.725,376.193,-79.768,-176.037,8.599,148.559
C08000=1185.721,376.441,-79.802,-176.035,8.602,148.559
C08001=1185.717,376.688,-79.837,-176.034,8.605,148.560
C08002=1185.713,376.936,-79.872,-176.033,8.609,148.560
C08003=1185.709,377.184,-79.907,-176.032,8.612,148.561
C08004=1185.705,377.431,-79.942,-176.031,8.615,148.561
C08005=1185.701,377.679,-79.976,-176.030,8.619,148.562
C08006=1185.697,377.926,-80.011,-176.028,8.622,148.562
C08007=1185.693,378.174,-80.046,-176.028,8.625,148.563
C08008=1185.688,378.421,-80.080,-176.026,8.629,148.564
C08009=1185.685,378.669,-80.116,-176.025,8.632,148.564
C08010=1185.681,378.916,-80.150,-176.024,8.635,148.565
C08011=1185.677,379.164,-80.185,-176.023,8.638,148.565
C08012=1185.673,379.411,-80.220,-176.022,8.642,148.566
C08013=1185.669,379.659,-80.255,-176.021,8.645,148.566
C08014=1185.665,379.906,-80.290,-176.020,8.648,148.567
C08015=1185.661,380.154,-80.325,-176.019,8.651,148.567
C08016=1185.657,380.402,-80.359,-176.018,8.655,148.568
C08017=1185.653,380.648,-80.394,-176.017,8.658,148.569
C08018=1185.649,380.897,-80.429,-176.016,8.661,148.569
C08019=1185.645,381.143,-80.464,-176.015,8.664,148.570
C08020=1185.641,381.391,-80.499,-176.014,8.667,148.570
C08021=1185.637,381.639,-80.534,-176.013,8.670,148.571
C08022=1185.633,381.886,-80.569,-176.012,8.673,148.571
C08023=1185.629,382.134,-80.604,-176.011,8.677,148.572
C08024=1185.624,382.381,-80.639,-176.010,8.680,148.573
C08025=1185.621,382.629,-80.673,-176.009,8.683,148.573
C08026=1185.617,382.877,-80.709,-176.009,8.686,148.574
C08027=1185.613,383.124,-80.743,-176.008,8.689,148.574
C08028=1185.609,383.371,-80.779,-176.007,8.692,148.575
C08029=1185.605,383.619,-80.813,-176.006,8.695,148.575
C08030=1185.601,383.866,-80.849,-176.005,8.699,148.576
C08031=1185.597,384.114,-80.884,-176.005,8.702,148.577
C08032=1185.593,384.361,-80.919,-176.004,8.705,148.577
C08033=1185.589,384.609,-80.954,-176.003,8.708,148.578
C08034=1185.585,384.857,-80.989,-176.002,8.711,148.578
C08035=1185.581,385.104,-81.024,-176.001,8.714,148.579
C08036=1185.577,385.352,-81.059,-176.001,8.716,148.579
C08037=1185.573,385.599,-81.094,-176.001,8.720,148.580
C08038=1185.569,385.846,-81.130,-176.000,8.723,148.581
C08039=1185.565,386.094,-81.165,-175.999,8.726,148.581
C08040=1185.561,386.341,-81.200,-175.998,8.729,148.582
C08041=1185.557,386.589,-81.235,-175.998,8.732,148.583
C08042=1185.553,386.837,-81.270,-175.997,8.734,148.583
C08043=1185.549,387.084,-81.305,-175.996,8.737,148.584
C08044=1185.545,387.332,-81.340,-175.996,8.741,148.584
C08045=1185.541,387.579,-81.376,-175.995,8.744,148.585
C08046=1185.537,387.826,-81.411,-175.995,8.746,148.586
C08047=1185.533,388.074,-81.446,-175.994,8.749,148.586
C08048=1185.529,388.322,-81.481,-175.993,8.752,148.587
C08049=1185.525,388.568,-81.517,-175.993,8.756,148.588
C08050=1185.521,388.816,-81.551,-175.993,8.758,148.588
C08051=1185.517,389.064,-81.587,-175.992,8.761,148.589
C08052=1185.513,389.311,-81.622,-175.992,8.763,148.589
C08053=1185.509,389.559,-81.657,-175.991,8.767,148.590
C08054=1185.506,389.806,-81.692,-175.991,8.770,148.591
C08055=1185.501,390.053,-81.728,-175.990,8.772,148.591
C08056=1185.497,390.301,-81.762,-175.990,8.776,148.592
C08057=1185.494,390.549,-81.798,-175.990,8.778,148.592
C08058=1185.489,390.796,-81.833,-175.989,8.781,148.593
C08059=1185.486,391.043,-81.869,-175.989,8.783,148.593
C08060=1185.482,391.291,-81.904,-175.988,8.787,148.594
C08061=1185.478,391.539,-81.939,-175.988,8.789,148.595
C08062=1185.474,391.822,-81.980,-175.988,8.792,148.596
C08063=1185.469,392.106,-82.020,-175.987,8.795,148.596
C08064=1185.465,392.390,-82.061,-175.986,8.799,148.597
C08065=1185.460,392.674,-82.101,-175.986,8.802,148.598
C08066=1185.455,392.921,-82.137,-175.986,8.804,148.598
C08067=1185.451,393.168,-82.172,-175.985,8.808,148.599
C08068=1185.447,393.416,-82.208,-175.985,8.810,148.600
C08069=1185.444,393.664,-82.243,-175.985,8.812,148.600
C08070=1185.440,393.911,-82.278,-175.985,8.816,148.601
C08071=1185.436,394.158,-82.313,-175.984,8.818,148.601
C08072=1185.432,394.406,-82.349,-175.984,8.820,148.602
C08073=1185.428,394.653,-82.384,-175.984,8.824,148.603
C08074=1185.424,394.901,-82.419,-175.983,8.826,148.603
C08075=1185.420,395.148,-82.454,-175.983,8.828,148.604
C08076=1185.416,395.396,-82.491,-175.983,8.832,148.605
C08077=1185.412,395.643,-82.526,-175.982,8.834,148.605
C08078=1185.408,395.890,-82.561,-175.983,8.836,148.606
C08079=1185.404,396.138,-82.597,-175.982,8.839,148.606
C08080=1185.400,396.385,-82.632,-175.982,8.842,148.607
C08081=1185.396,396.633,-82.667,-175.982,8.844,148.608
C08082=1185.392,396.880,-82.702,-175.982,8.847,148.608
C08083=1185.388,397.128,-82.738,-175.981,8.849,148.609
C08084=1185.384,397.375,-82.774,-175.981,8.851,148.609
C08085=1185.380,397.623,-82.810,-175.981,8.855,148.610
C08086=1185.376,397.870,-82.845,-175.981,8.857,148.611
C08087=1185.372,398.117,-82.880,-175.981,8.859,148.611
C08088=1185.369,398.365,-82.916,-175.980,8.862,148.612
C08089=1185.364,398.612,-82.952,-175.981,8.864,148.612
C08090=1185.360,398.859,-82.987,-175.980,8.866,148.613
C08091=1185.356,399.107,-83.022,-175.980,8.869,148.613
C08092=1185.353,399.355,-83.058,-175.980,8.872,148.614
C08093=1185.349,399.602,-83.093,-175.979,8.874,148.615
C08094=1185.344,399.849,-83.129,-175.980,8.877,148.616
C08095=1185.340,400.097,-83.164,-175.979,8.879,148.616
C08096=1185.337,400.344,-83.200,-175.979,8.881,148.617
C08097=1185.333,400.592,-83.236,-175.979,8.884,148.617
C08098=1185.329,400.839,-83.271,-175.979,8.886,148.618
C08099=1185.324,401.087,-83.307,-175.979,8.889,148.618
C08100=1185.321,401.334,-83.342,-175.979,8.891,148.619
C08101=1185.317,401.582,-83.378,-175.979,8.893,148.620
C08102=1185.313,401.829,-83.414,-175.979,8.896,148.620
C08103=1185.309,402.076,-83.449,-175.979,8.898,148.621
C08104=1185.305,402.324,-83.485,-175.978,8.901,148.621
C08105=1185.301,402.571,-83.520,-175.978,8.903,148.622
C08106=1185.297,402.819,-83.556,-175.978,8.905,148.623
C08107=1185.294,403.066,-83.591,-175.978,8.908,148.623
C08108=1185.289,403.313,-83.627,-175.978,8.910,148.624
C08109=1185.285,403.561,-83.663,-175.978,8.912,148.624
C08110=1185.281,403.808,-83.698,-175.978,8.915,148.625
C08111=1185.278,404.056,-83.734,-175.978,8.916,148.626
C08112=1185.274,404.303,-83.769,-175.978,8.919,148.626
C08113=1185.269,404.550,-83.805,-175.978,8.921,148.627
C08114=1185.265,404.798,-83.841,-175.978,8.924,148.627
C08115=1185.262,405.045,-83.876,-175.978,8.926,148.628
C08116=1185.258,405.293,-83.912,-175.978,8.928,148.628
C08117=1185.254,405.541,-83.948,-175.978,8.931,148.629
C08118=1185.249,405.787,-83.983,-175.977,8.933,148.630
C08119=1185.246,406.035,-84.019,-175.978,8.934,148.630
C08120=1185.242,406.282,-84.054,-175.978,8.937,148.631
C08121=1185.238,406.530,-84.090,-175.978,8.939,148.631
C08122=1185.234,406.778,-84.126,-175.977,8.941,148.632
C08123=1185.230,407.025,-84.161,-175.977,8.944,148.632
C08124=1185.226,407.271,-84.197,-175.977,8.946,148.633
C08125=1185.222,407.519,-84.234,-175.978,8.948,148.634
C08126=1185.218,407.767,-84.269,-175.977,8.950,148.634
C08127=1185.215,408.014,-84.305,-175.977,8.952,148.635
C08128=1185.210,408.261,-84.340,-175.977,8.955,148.635
C08129=1185.206,408.509,-84.376,-175.978,8.956,148.636
C08130=1185.202,408.756,-84.412,-175.977,8.959,148.636
C08131=1185.199,409.004,-84.447,-175.977,8.961,148.637
C08132=1185.194,409.252,-84.483,-175.977,8.963,148.638
C08133=1185.190,409.499,-84.519,-175.978,8.965,148.638
C08134=1185.187,409.745,-84.555,-175.977,8.967,148.639
C08135=1185.182,409.993,-84.591,-175.977,8.969,148.639
C08136=1185.178,410.241,-84.626,-175.977,8.972,148.640
C08137=1185.175,410.488,-84.662,-175.978,8.973,148.640
C08138=1185.171,410.736,-84.697,-175.977,8.976,148.641
C08139=1185.167,410.984,-84.734,-175.977,8.978,148.641
C08140=1185.162,411.230,-84.769,-175.977,8.979,148.642
C08141=1185.159,411.478,-84.804,-175.977,8.982,148.642
C08142=1185.155,411.725,-84.841,-175.977,8.984,148.643
C08143=1185.151,411.973,-84.877,-175.978,8.986,148.643
C08144=1185.147,412.220,-84.912,-175.977,8.988,148.644
C08145=1185.143,412.468,-84.948,-175.977,8.990,148.644
C08146=1185.139,412.715,-84.984,-175.977,8.992,148.645
C08147=1185.135,412.962,-85.019,-175.977,8.994,148.645
C08148=1185.131,413.209,-85.056,-175.977,8.996,148.646
C08149=1185.127,413.457,-85.092,-175.978,8.998,148.647
C08150=1185.124,413.704,-85.127,-175.977,9.000,148.647
C08151=1185.119,413.952,-85.163,-175.978,9.001,148.648
C08152=1185.116,414.200,-85.199,-175.977,9.004,148.648
C08153=1185.111,414.446,-85.234,-175.977,9.006,148.649
C08154=1185.107,414.694,-85.271,-175.977,9.007,148.649
C08155=1185.104,414.941,-85.306,-175.977,9.010,148.650
C08156=1185.100,415.189,-85.342,-175.977,9.012,148.650
C08157=1185.095,415.436,-85.378,-175.977,9.013,148.651
C08158=1185.093,415.648,-85.408,-175.977,9.015,148.651
C08159=1185.089,415.860,-85.439,-175.977,9.017,148.652
C08160=1185.087,416.072,-85.470,-175.977,9.019,148.652
C08161=1185.085,416.284,-85.501,-175.977,9.020,148.652
C08162=1185.085,416.495,-85.530,-175.977,9.022,148.653
C08163=1185.085,416.707,-85.561,-175.977,9.023,148.653
C08164=1185.086,416.919,-85.592,-175.977,9.024,148.654
C08165=1185.088,417.130,-85.621,-175.977,9.027,148.654
C08166=1184.667,417.131,-85.663,-175.980,9.037,148.658
C08167=1184.665,416.918,-85.633,-175.981,9.035,148.657
C08168=1184.664,416.705,-85.603,-175.980,9.034,148.657
C08169=1184.663,416.492,-85.571,-175.980,9.033,148.656
C08170=1184.664,416.279,-85.541,-175.980,9.031,148.656
C08171=1184.665,416.065,-85.510,-175.981,9.029,148.656
C08172=1184.668,415.852,-85.480,-175.980,9.028,148.655
C08173=1184.670,415.638,-85.449,-175.980,9.027,148.655
C08174=1184.675,415.425,-85.418,-175.981,9.024,148.654
C08175=1184.678,415.177,-85.382,-175.980,9.023,148.654
C08176=1184.682,414.931,-85.347,-175.981,9.021,148.653
C08177=1184.687,414.683,-85.310,-175.980,9.018,148.653
C08178=1184.690,414.436,-85.274,-175.980,9.017,148.652
C08179=1184.694,414.188,-85.239,-175.980,9.014,148.652
C08180=1184.698,413.941,-85.203,-175.980,9.013,148.651
C08181=1184.702,413.693,-85.167,-175.980,9.011,148.651
C08182=1184.705,413.446,-85.131,-175.981,9.008,148.650
C08183=1184.710,413.199,-85.095,-175.980,9.007,148.650
C08184=1184.714,412.952,-85.060,-175.981,9.005,148.649
C08185=1184.718,412.704,-85.024,-175.980,9.002,148.649
C08186=1184.722,412.456,-84.988,-175.980,9.001,148.648
C08187=1184.726,412.209,-84.952,-175.980,8.998,148.648
C08188=1184.729,411.962,-84.916,-175.981,8.996,148.647
C08189=1184.733,411.714,-84.880,-175.980,8.995,148.647
C08190=1184.738,411.467,-84.845,-175.981,8.993,148.646
C08191=1184.741,411.220,-84.809,-175.980,8.990,148.645
C08192=1184.746,410.972,-84.773,-175.980,8.989,148.645
C08193=1184.749,410.724,-84.738,-175.980,8.986,148.644
C08194=1184.753,410.477,-84.702,-175.981,8.984,148.644
C08195=1184.757,410.230,-84.665,-175.980,8.983,148.643
C08196=1184.761,409.983,-84.630,-175.980,8.980,148.643
C08197=1184.765,409.735,-84.594,-175.980,8.978,148.642
C08198=1184.769,409.488,-84.559,-175.980,8.976,148.642
C08199=1184.773,409.240,-84.523,-175.980,8.974,148.641
C08200=1184.777,408.993,-84.487,-175.980,8.971,148.640
C08201=1184.780,408.745,-84.452,-175.980,8.969,148.640
C08202=1184.785,408.498,-84.416,-175.980,8.968,148.639
C08203=1184.789,408.251,-84.380,-175.980,8.965,148.639
C08204=1184.793,408.004,-84.344,-175.980,8.963,148.638
C08205=1184.796,407.756,-84.308,-175.980,8.961,148.638
C08206=1184.801,407.508,-84.272,-175.980,8.959,148.637
C08207=1184.804,407.261,-84.237,-175.980,8.957,148.637
C08208=1184.809,407.014,-84.202,-175.980,8.954,148.636
C08209=1184.813,406.766,-84.165,-175.980,8.952,148.635
C08210=1184.817,406.519,-84.130,-175.981,8.950,148.635
C08211=1184.820,406.271,-84.094,-175.980,8.948,148.634
C08212=1184.824,406.024,-84.059,-175.980,8.946,148.634
C08213=1184.829,405.777,-84.023,-175.981,8.944,148.633
C08214=1184.833,405.529,-83.987,-175.980,8.941,148.633
C08215=1184.836,405.282,-83.952,-175.981,8.939,148.632
C08216=1184.840,405.035,-83.916,-175.981,8.936,148.631
C08217=1184.844,404.787,-83.880,-175.980,8.935,148.631
C08218=1184.848,404.539,-83.844,-175.980,8.932,148.630
C08219=1184.852,404.293,-83.809,-175.981,8.930,148.630
C08220=1184.856,404.045,-83.773,-175.980,8.928,148.629
C08221=1184.860,403.797,-83.737,-175.981,8.925,148.629
C08222=1184.864,403.550,-83.702,-175.981,8.923,148.628
C08223=1184.867,403.302,-83.666,-175.981,8.921,148.627
C08224=1184.872,403.056,-83.631,-175.981,8.918,148.627
C08225=1184.876,402.808,-83.595,-175.981,8.916,148.626
C08226=1184.880,402.560,-83.559,-175.981,8.913,148.626
C08227=1184.883,402.313,-83.524,-175.981,8.911,148.625
C08228=1184.888,402.066,-83.488,-175.982,8.909,148.624
C08229=1184.892,401.818,-83.452,-175.981,8.906,148.624
C08230=1184.896,401.571,-83.417,-175.982,8.904,148.623
C08231=1184.899,401.323,-83.381,-175.982,8.902,148.622
C08232=1184.903,401.076,-83.346,-175.982,8.899,148.622
C08233=1184.907,400.829,-83.310,-175.982,8.897,148.621
C08234=1184.912,400.581,-83.274,-175.982,8.894,148.621
C08235=1184.915,400.333,-83.239,-175.982,8.892,148.620
C08236=1184.919,400.086,-83.203,-175.982,8.890,148.620
C08237=1184.923,399.839,-83.168,-175.982,8.887,148.619
C08238=1184.927,399.592,-83.132,-175.982,8.885,148.618
C08239=1184.932,399.343,-83.097,-175.982,8.883,148.618
C08240=1184.935,399.096,-83.061,-175.983,8.880,148.617
C08241=1184.939,398.848,-83.026,-175.983,8.878,148.617
C08242=1184.943,398.601,-82.991,-175.983,8.875,148.616
C08243=1184.947,398.354,-82.955,-175.983,8.873,148.615
C08244=1184.950,398.106,-82.920,-175.983,8.871,148.615
C08245=1184.955,397.859,-82.884,-175.983,8.867,148.614
C08246=1184.959,397.612,-82.848,-175.984,8.865,148.614
C08247=1184.963,397.364,-82.813,-175.984,8.863,148.613
C08248=1184.966,397.117,-82.777,-175.984,8.860,148.612
C08249=1184.970,396.869,-82.742,-175.984,8.858,148.612
C08250=1184.974,396.623,-82.707,-175.984,8.856,148.611
C08251=1184.979,396.374,-82.671,-175.985,8.852,148.611
C08252=1184.983,396.127,-82.636,-175.985,8.850,148.610
C08253=1184.986,395.879,-82.600,-175.985,8.848,148.609
C08254=1184.991,395.632,-82.565,-175.985,8.845,148.609
C08255=1184.994,395.385,-82.529,-175.985,8.842,148.608
C08256=1184.998,395.137,-82.494,-175.986,8.840,148.607
C08257=1185.003,394.890,-82.458,-175.985,8.837,148.607
C08258=1185.007,394.642,-82.423,-175.986,8.834,148.606
C08259=1185.011,394.395,-82.388,-175.987,8.832,148.606
C08260=1185.014,394.147,-82.352,-175.986,8.829,148.605
C08261=1185.019,393.900,-82.317,-175.987,8.826,148.604
C08262=1185.022,393.653,-82.281,-175.987,8.824,148.604
C08263=1185.026,393.405,-82.246,-175.987,8.821,148.603
C08264=1185.030,393.157,-82.211,-175.988,8.818,148.602
C08265=1185.034,392.910,-82.176,-175.988,8.816,148.602
C08266=1185.039,392.663,-82.140,-175.989,8.813,148.601
C08267=1185.043,392.379,-82.099,-175.988,8.810,148.600
C08268=1185.048,392.095,-82.059,-175.989,8.807,148.600
C08269=1185.052,391.812,-82.018,-175.990,8.803,148.599
C08270=1185.056,391.527,-81.978,-175.990,8.800,148.598
C08271=1185.060,391.280,-81.942,-175.990,8.798,148.598
C08272=1185.064,391.033,-81.907,-175.991,8.794,148.597
C08273=1185.068,390.785,-81.872,-175.991,8.792,148.596
C08274=1185.072,390.538,-81.837,-175.992,8.789,148.596
C08275=1185.076,390.290,-81.801,-175.992,8.787,148.595
C08276=1185.080,390.043,-81.766,-175.992,8.783,148.595
C08277=1185.084,389.795,-81.731,-175.993,8.780,148.594
C08278=1185.088,389.548,-81.696,-175.993,8.778,148.593
C08279=1185.092,389.300,-81.660,-175.994,8.775,148.593
C08280=1185.096,389.052,-81.625,-175.994,8.772,148.592
C08281=1185.100,388.806,-81.590,-175.995,8.769,148.592
C08282=1185.103,388.558,-81.555,-175.996,8.766,148.591
C08283=1185.107,388.311,-81.519,-175.996,8.764,148.590
C08284=1185.112,388.063,-81.485,-175.996,8.760,148.590
C08285=1185.116,387.815,-81.448,-175.997,8.757,148.589
C08286=1185.120,387.568,-81.413,-175.998,8.754,148.589
C08287=1185.124,387.320,-81.378,-175.998,8.752,148.588
C08288=1185.128,387.073,-81.343,-175.999,8.749,148.587
C08289=1185.132,386.825,-81.308,-175.999,8.746,148.587
C08290=1185.136,386.578,-81.273,-176.000,8.742,148.586
C08291=1185.140,386.330,-81.237,-176.000,8.740,148.586
C08292=1185.144,386.082,-81.202,-176.001,8.737,148.585
C08293=1185.147,385.836,-81.168,-176.002,8.734,148.584
C08294=1185.151,385.588,-81.132,-176.002,8.731,148.584
C08295=1185.155,385.340,-81.097,-176.003,8.727,148.583
C08296=1185.159,385.093,-81.062,-176.004,8.724,148.582
C08297=1185.163,384.845,-81.027,-176.005,8.721,148.582
C08298=1185.168,384.598,-80.992,-176.006,8.718,148.581
C08299=1185.171,384.351,-80.957,-176.007,8.715,148.581
C08300=1185.175,384.103,-80.922,-176.007,8.713,148.580
C08301=1185.179,383.856,-80.887,-176.008,8.710,148.580
C08302=1185.183,383.608,-80.852,-176.008,8.707,148.579
C08303=1185.187,383.360,-80.816,-176.009,8.704,148.578
C08304=1185.192,383.113,-80.782,-176.010,8.700,148.578
C08305=1185.195,382.866,-80.746,-176.011,8.697,148.577
C08306=1185.200,382.618,-80.712,-176.012,8.693,148.577
C08307=1185.204,382.371,-80.676,-176.013,8.690,148.576
C08308=1185.207,382.122,-80.641,-176.014,8.687,148.575
C08309=1185.212,381.876,-80.606,-176.015,8.684,148.575
C08310=1185.215,381.628,-80.572,-176.015,8.681,148.574
C08311=1185.219,381.381,-80.537,-176.016,8.678,148.574
C08312=1185.223,381.133,-80.502,-176.017,8.675,148.573
C08313=1185.227,380.885,-80.466,-176.018,8.672,148.573
C08314=1185.231,380.638,-80.432,-176.019,8.668,148.572
C08315=1185.235,380.390,-80.397,-176.020,8.665,148.571
C08316=1185.240,380.143,-80.362,-176.021,8.662,148.571
C08317=1185.244,379.895,-80.327,-176.022,8.659,148.570
C08318=1185.248,379.648,-80.292,-176.023,8.656,148.570
C08319=1185.251,379.400,-80.258,-176.024,8.652,148.569
C08320=1185.255,379.152,-80.223,-176.025,8.649,148.569
C08321=1185.259,378.905,-80.188,-176.026,8.646,148.568
C08322=1185.263,378.657,-80.153,-176.027,8.643,148.568
C08323=1185.268,378.411,-80.118,-176.029,8.639,148.567
C08324=1185.272,378.162,-80.083,-176.029,8.636,148.566
C08325=1185.275,377.915,-80.049,-176.031,8.633,148.566
C08326=1185.279,377.668,-80.013,-176.032,8.629,148.565
C08327=1185.284,377.420,-79.979,-176.033,8.626,148.565
C08328=1185.288,377.172,-79.944,-176.034,8.623,148.564
C08329=1185.292,376.925,-79.909,-176.035,8.619,148.564
C08330=1185.295,376.678,-79.875,-176.036,8.616,148.563
C08331=1185.299,376.430,-79.840,-176.038,8.613,148.563
C08332=1185.304,376.182,-79.805,-176.039,8.609,148.562
C08333=1185.307,375.935,-79.770,-176.040,8.606,148.562
C08334=1185.311,375.688,-79.736,-176.041,8.603,148.561
C08335=1185.315,375.439,-79.701,-176.042,8.600,148.560
C08336=1185.320,375.192,-79.667,-176.044,8.596,148.560
C08337=1185.323,374.944,-79.631,-176.045,8.593,148.559
C08338=1185.327,374.697,-79.597,-176.047,8.589,148.559
C08339=1185.331,374.449,-79.562,-176.047,8.586,148.558
C08340=1185.336,374.202,-79.528,-176.049,8.583,148.558
C08341=1185.340,373.954,-79.493,-176.050,8.580,148.557
C08342=1185.343,373.707,-79.459,-176.052,8.576,148.557
C08343=1185.347,373.459,-79.424,-176.053,8.573,148.556
C08344=1185.352,373.212,-79.389,-176.055,8.569,148.556
C08345=1185.355,372.964,-79.355,-176.056,8.566,148.556
C08346=1185.360,372.716,-79.321,-176.057,8.562,148.555
C08347=1185.364,372.468,-79.286,-176.058,8.560,148.555
C08348=1185.367,372.221,-79.252,-176.060,8.556,148.554
C08349=1185.372,371.974,-79.217,-176.062,8.552,148.554
C08350=1185.376,371.726,-79.182,-176.063,8.549,148.553
C08351=1185.379,371.479,-79.148,-176.064,8.545,148.552
C08352=1185.383,371.231,-79.113,-176.065,8.543,148.552
C08353=1185.388,370.984,-79.079,-176.067,8.539,148.552
C08354=1185.391,370.736,-79.044,-176.069,8.535,148.551
C08355=1185.396,370.488,-79.010,-176.070,8.532,148.551
C08356=1185.399,370.241,-78.976,-176.072,8.529,148.550
C08357=1185.404,369.993,-78.941,-176.073,8.525,148.550
C08358=1185.408,369.746,-78.907,-176.075,8.522,148.549
C08359=1185.411,369.498,-78.873,-176.077,8.519,148.549
C08360=1185.416,369.251,-78.838,-176.078,8.515,148.548
C08361=1185.419,369.003,-78.804,-176.079,8.512,148.548
C08362=1185.424,368.755,-78.769,-176.081,8.508,148.548
C08363=1185.428,368.508,-78.735,-176.083,8.505,148.547
C08364=1185.432,368.260,-78.701,-176.085,8.501,148.547
C08365=1185.436,368.013,-78.666,-176.086,8.498,148.546
C08366=1185.440,367.764,-78.633,-176.088,8.495,148.546
C08367=1185.444,367.517,-78.598,-176.089,8.491,148.545
C08368=1185.448,367.270,-78.564,-176.091,8.488,148.545
C08369=1185.452,367.022,-78.530,-176.093,8.485,148.545
C08370=1185.456,366.774,-78.496,-176.094,8.481,148.544
C08371=1185.461,366.493,-78.456,-176.096,8.477,148.544
C08372=1185.465,366.212,-78.417,-176.098,8.473,148.543
C08373=1185.470,365.931,-78.379,-176.100,8.469,148.543
C08374=1185.475,365.649,-78.340,-176.102,8.465,148.542
C08375=1185.478,365.401,-78.306,-176.104,8.462,148.542
C08376=1185.483,365.153,-78.271,-176.105,8.458,148.541
C08377=1185.486,364.906,-78.238,-176.107,8.454,148.541
C08378=1185.491,364.658,-78.203,-176.109,8.452,148.541
C08379=1185.495,364.410,-78.170,-176.111,8.448,148.540
C08380=1185.498,364.163,-78.136,-176.112,8.445,148.540
C08381=1185.502,363.915,-78.101,-176.114,8.441,148.539
C08382=1185.506,363.667,-78.068,-176.116,8.437,148.539
C08383=1185.511,363.420,-78.033,-176.118,8.434,148.539
C08384=1185.514,363.172,-77.999,-176.120,8.431,148.538
C08385=1185.518,362.925,-77.965,-176.121,8.428,148.538
C08386=1185.523,362.677,-77.931,-176.123,8.424,148.537
C08387=1185.526,362.429,-77.897,-176.125,8.420,148.537
C08388=1185.531,362.182,-77.863,-176.127,8.417,148.537
C08389=1185.535,361.934,-77.830,-176.129,8.414,148.536
C08390=1185.538,361.686,-77.795,-176.131,8.410,148.536
C08391=1185.543,361.438,-77.762,-176.133,8.407,148.536
C08392=1185.547,361.191,-77.728,-176.135,8.403,148.535
C08393=1185.551,360.944,-77.694,-176.136,8.400,148.535
C08394=1185.555,360.695,-77.660,-176.138,8.397,148.535
C08395=1185.559,360.448,-77.626,-176.140,8.393,148.534
C08396=1185.563,360.201,-77.593,-176.142,8.390,148.534
C08397=1185.567,359.953,-77.558,-176.144,8.386,148.534
C08398=1185.571,359.705,-77.525,-176.146,8.383,148.533
C08399=1185.575,359.458,-77.491,-176.148,8.379,148.533
C08400=1185.580,359.210,-77.457,-176.150,8.376,148.533
C08401=1185.584,358.962,-77.423,-176.152,8.372,148.532
C08402=1185.587,358.714,-77.390,-176.154,8.369,148.532
C08403=1185.591,358.467,-77.356,-176.156,8.365,148.532
C08404=1185.596,358.219,-77.322,-176.158,8.362,148.531
C08405=1185.600,357.972,-77.288,-176.161,8.358,148.531
C08406=1185.603,357.723,-77.255,-176.162,8.355,148.531
C08407=1185.607,357.476,-77.221,-176.165,8.352,148.530
C08408=1185.612,357.228,-77.187,-176.167,8.348,148.530
C08409=1185.616,356.980,-77.154,-176.169,8.345,148.530
C08410=1185.620,356.733,-77.120,-176.171,8.341,148.529
C08411=1185.623,356.485,-77.086,-176.173,8.338,148.529
C08412=1185.628,356.237,-77.053,-176.175,8.334,148.529
C08413=1185.632,355.990,-77.019,-176.177,8.331,148.529
C08414=1185.636,355.742,-76.986,-176.179,8.327,148.528
C08415=1185.640,355.494,-76.953,-176.181,8.325,148.528
C08416=1185.644,355.247,-76.919,-176.183,8.322,148.528
C08417=1185.648,354.999,-76.885,-176.185,8.318,148.527
C08418=1185.652,354.751,-76.852,-176.187,8.315,148.527
C08419=1185.656,354.504,-76.818,-176.189,8.311,148.527
C08420=1185.661,354.256,-76.784,-176.191,8.308,148.526
C08421=1185.665,354.008,-76.751,-176.193,8.304,148.526
C08422=1185.669,353.760,-76.718,-176.196,8.301,148.526
C08423=1185.673,353.513,-76.684,-176.198,8.298,148.526
C08424=1185.676,353.265,-76.651,-176.200,8.294,148.525
C08425=1185.680,353.017,-76.618,-176.202,8.291,148.525
C08426=1185.685,352.769,-76.584,-176.204,8.287,148.525
C08427=1185.689,352.522,-76.551,-176.206,8.284,148.525
C08428=1185.694,352.274,-76.517,-176.208,8.281,148.524
C08429=1185.697,352.027,-76.484,-176.210,8.277,148.524
C08430=1185.701,351.779,-76.450,-176.213,8.274,148.524
C08431=1185.706,351.531,-76.417,-176.215,8.271,148.524
C08432=1185.710,351.283,-76.384,-176.217,8.267,148.523
C08433=1185.714,351.036,-76.351,-176.219,8.264,148.523
C08434=1185.717,350.787,-76.317,-176.221,8.260,148.523
C08435=1185.722,350.539,-76.284,-176.224,8.257,148.522
C08436=1185.726,350.292,-76.251,-176.226,8.254,148.522
C08437=1185.730,350.044,-76.218,-176.228,8.250,148.522
C08438=1185.734,349.796,-76.185,-176.230,8.247,148.522
C08439=1185.738,349.549,-76.152,-176.232,8.243,148.521
C08440=1185.742,349.301,-76.119,-176.234,8.240,148.521
C08441=1185.746,349.053,-76.085,-176.237,8.237,148.521
C08442=1185.751,348.805,-76.052,-176.239,8.233,148.521
C08443=1185.755,348.558,-76.019,-176.241,8.230,148.520
C08444=1185.759,348.310,-75.986,-176.243,8.228,148.520
C08445=1185.763,348.062,-75.953,-176.245,8.224,148.520
C08446=1185.767,347.814,-75.920,-176.247,8.221,148.520
C08447=1185.771,347.567,-75.886,-176.250,8.218,148.520
C08448=1185.775,347.319,-75.854,-176.252,8.214,148.519
C08449=1185.779,347.072,-75.821,-176.254,8.211,148.519
C08450=1185.783,346.823,-75.788,-176.256,8.208,148.519
C08451=1185.787,346.575,-75.755,-176.259,8.204,148.519
C08452=1185.792,346.328,-75.722,-176.261,8.201,148.519
C08453=1185.796,346.080,-75.689,-176.263,8.198,148.518
C08454=1185.800,345.832,-75.656,-176.265,8.194,148.518
C08455=1185.804,345.585,-75.622,-176.268,8.191,148.518
C08456=1185.808,345.336,-75.590,-176.270,8.188,148.518
C08457=1185.812,345.089,-75.557,-176.272,8.184,148.517
C08458=1185.816,344.841,-75.524,-176.274,8.181,148.517
C08459=1185.820,344.593,-75.491,-176.277,8.178,148.517
C08460=1185.824,344.345,-75.459,-176.279,8.175,148.517
C08461=1185.829,344.097,-75.426,-176.281,8.171,148.517
C08462=1185.833,343.849,-75.392,-176.283,8.168,148.516
C08463=1185.836,343.602,-75.360,-176.286,8.165,148.516
C08464=1185.841,343.354,-75.327,-176.287,8.162,148.516
C08465=1185.845,343.107,-75.295,-176.290,8.159,148.516
C08466=1185.849,342.859,-75.261,-176.292,8.155,148.516
C08467=1185.854,342.611,-75.229,-176.294,8.152,148.515
C08468=1185.857,342.363,-75.196,-176.296,8.149,148.515
C08469=1185.861,342.115,-75.163,-176.299,8.145,148.515
C08470=1185.866,341.867,-75.131,-176.301,8.142,148.515
C08471=1185.870,341.619,-75.098,-176.304,8.139,148.515
C08472=1185.874,341.371,-75.066,-176.306,8.136,148.514
C08473=1185.878,341.124,-75.033,-176.308,8.133,148.514
C08474=1185.882,340.875,-75.000,-176.310,8.129,148.514
C08475=1185.887,340.597,-74.964,-176.313,8.126,148.514
C08476=1185.891,340.318,-74.927,-176.315,8.122,148.514
C08477=1185.896,340.039,-74.890,-176.318,8.118,148.513
C08478=1185.901,339.761,-74.853,-176.321,8.115,148.513
C08479=1185.905,339.512,-74.821,-176.323,8.111,148.513
C08480=1185.909,339.265,-74.788,-176.325,8.108,148.513
C08481=1185.913,339.017,-74.756,-176.327,8.105,148.513
C08482=1185.917,338.770,-74.724,-176.329,8.102,148.512
C08483=1185.922,338.522,-74.691,-176.332,8.099,148.512
C08484=1185.926,338.274,-74.658,-176.334,8.096,148.512
C08485=1185.929,338.026,-74.626,-176.337,8.092,148.512
C08486=1185.934,337.777,-74.594,-176.339,8.089,148.512
C08487=1185.938,337.530,-74.561,-176.341,8.086,148.512
C08488=1185.942,337.282,-74.529,-176.344,8.083,148.512
C08489=1185.947,337.034,-74.497,-176.346,8.080,148.511
C08490=1185.950,336.787,-74.464,-176.348,8.076,148.511
C08491=1185.955,336.538,-74.432,-176.351,8.073,148.511
C08492=1185.958,336.290,-74.400,-176.353,8.070,148.511
C08493=1185.963,336.043,-74.367,-176.355,8.067,148.511
C08494=1185.967,335.795,-74.335,-176.358,8.063,148.511
C08495=1185.971,335.547,-74.303,-176.360,8.061,148.511
C08496=1185.975,335.299,-74.270,-176.362,8.058,148.510
C08497=1185.979,335.051,-74.238,-176.364,8.054,148.510
C08498=1185.983,334.804,-74.206,-176.367,8.051,148.510
C08499=1185.988,334.555,-74.174,-176.369,8.048,148.510
C08500=1185.991,334.308,-74.141,-176.372,8.045,148.510
C08501=1185.996,334.060,-74.109,-176.374,8.041,148.510
C08502=1186.000,333.812,-74.077,-176.377,8.038,148.510
C08503=1186.004,333.564,-74.045,-176.379,8.035,148.509
C08504=1186.008,333.316,-74.013,-176.381,8.032,148.509
C08505=1186.012,333.068,-73.980,-176.384,8.029,148.509
C08506=1186.017,332.821,-73.949,-176.386,8.025,148.509
C08507=1186.021,332.572,-73.916,-176.388,8.023,148.509
C08508=1186.025,332.324,-73.884,-176.390,8.020,148.509
C08509=1186.030,332.077,-73.852,-176.393,8.017,148.508
C08510=1186.034,331.829,-73.820,-176.395,8.013,148.508
C08511=1186.037,331.581,-73.789,-176.398,8.010,148.508
C08512=1186.042,331.332,-73.756,-176.400,8.007,148.508
C08513=1186.046,331.085,-73.725,-176.402,8.004,148.508
C08514=1186.050,330.837,-73.692,-176.405,8.001,148.508
C08515=1186.054,330.589,-73.660,-176.407,7.997,148.508
C08516=1186.058,330.341,-73.629,-176.410,7.994,148.508
C08517=1186.063,330.093,-73.596,-176.412,7.991,148.507
C08518=1186.067,329.845,-73.565,-176.414,7.988,148.507
C08519=1186.071,329.598,-73.533,-176.416,7.986,148.507
C08520=1186.075,329.349,-73.501,-176.419,7.982,148.507
C08521=1186.079,329.101,-73.469,-176.421,7.979,148.507
C08522=1186.083,328.854,-73.437,-176.424,7.976,148.507
C08523=1186.088,328.605,-73.405,-176.426,7.973,148.507
C08524=1186.091,328.357,-73.373,-176.429,7.970,148.507
C08525=1186.096,328.110,-73.342,-176.431,7.966,148.506
C08526=1186.099,327.862,-73.310,-176.434,7.963,148.506
C08527=1186.105,327.614,-73.278,-176.436,7.960,148.506
C08528=1186.108,327.366,-73.246,-176.439,7.957,148.506
C08529=1186.112,327.118,-73.215,-176.440,7.954,148.506
C08530=1186.117,326.870,-73.183,-176.443,7.951,148.506
C08531=1186.121,326.622,-73.151,-176.445,7.948,148.506
C08532=1186.125,326.375,-73.119,-176.448,7.945,148.506
C08533=1186.129,326.127,-73.087,-176.450,7.942,148.506
C08534=1186.133,325.878,-73.056,-176.453,7.939,148.506
C08535=1186.138,325.630,-73.024,-176.455,7.935,148.505
C08536=1186.142,325.382,-72.992,-176.458,7.932,148.505
C08537=1186.146,325.135,-72.961,-176.460,7.929,148.505
C08538=1186.150,324.886,-72.930,-176.463,7.926,148.505
C08539=1186.154,324.638,-72.898,-176.464,7.924,148.505
C08540=1186.158,324.391,-72.866,-176.467,7.921,148.505
C08541=1186.163,324.143,-72.834,-176.469,7.917,148.505
C08542=1186.167,323.895,-72.803,-176.472,7.914,148.505
C08543=1186.171,323.647,-72.771,-176.474,7.911,148.505
C08544=1186.175,323.399,-72.740,-176.477,7.908,148.505
C08545=1186.179,323.151,-72.709,-176.479,7.905,148.505
C08546=1186.184,322.903,-72.677,-176.482,7.902,148.505
C08547=1186.188,322.655,-72.646,-176.484,7.898,148.504
C08548=1186.191,322.407,-72.614,-176.486,7.896,148.504
C08549=1186.196,322.159,-72.583,-176.489,7.893,148.504
C08550=1186.200,321.911,-72.552,-176.491,7.890,148.504
C08551=1186.205,321.663,-72.520,-176.494,7.887,148.504
C08552=1186.209,321.414,-72.488,-176.496,7.884,148.504
C08553=1186.213,321.167,-72.457,-176.499,7.881,148.504
C08554=1186.217,320.918,-72.426,-176.501,7.877,148.504
C08555=1186.221,320.671,-72.394,-176.504,7.874,148.504
C08556=1186.225,320.422,-72.363,-176.506,7.871,148.504
C08557=1186.230,320.175,-72.332,-176.508,7.869,148.504
C08558=1186.234,319.926,-72.301,-176.511,7.866,148.504
C08559=1186.238,319.679,-72.269,-176.513,7.862,148.503
C08560=1186.242,319.431,-72.238,-176.516,7.859,148.503
C08561=1186.246,319.183,-72.207,-176.518,7.856,148.503
C08562=1186.251,318.935,-72.176,-176.521,7.853,148.503
C08563=1186.255,318.687,-72.144,-176.524,7.850,148.503
C08564=1186.259,318.439,-72.113,-176.526,7.847,148.503
C08565=1186.263,318.190,-72.082,-176.528,7.845,148.503
C08566=1186.267,317.943,-72.051,-176.530,7.841,148.503
C08567=1186.271,317.695,-72.020,-176.533,7.838,148.503
C08568=1186.275,317.447,-71.989,-176.536,7.835,148.503
C08569=1186.280,317.199,-71.958,-176.538,7.832,148.503
C08570=1186.284,316.951,-71.927,-176.541,7.829,148.503
C08571=1186.288,316.703,-71.896,-176.544,7.826,148.503
C08572=1186.292,316.455,-71.864,-176.545,7.823,148.503
C08573=1186.297,316.207,-71.833,-176.548,7.820,148.503
C08574=1186.301,315.959,-71.803,-176.551,7.817,148.503
C08575=1186.305,315.710,-71.771,-176.553,7.814,148.502
C08576=1186.309,315.463,-71.741,-176.556,7.811,148.502
C08577=1186.313,315.214,-71.709,-176.558,7.808,148.502
C08578=1186.317,314.966,-71.679,-176.561,7.805,148.502
C08579=1186.322,314.690,-71.643,-176.563,7.802,148.502
C08580=1186.327,314.413,-71.610,-176.566,7.799,148.502
C08581=1186.332,314.137,-71.575,-176.569,7.795,148.502
C08582=1186.336,313.860,-71.541,-176.572,7.792,148.502
C08583=1186.340,313.612,-71.510,-176.574,7.789,148.502
C08584=1186.345,313.364,-71.479,-176.577,7.786,148.502
C08585=1186.349,313.116,-71.448,-176.579,7.783,148.502
C08586=1186.354,312.868,-71.417,-176.581,7.780,148.502
C08587=1186.357,312.620,-71.387,-176.584,7.777,148.502
C08588=1186.362,312.371,-71.356,-176.586,7.774,148.502
C08589=1186.366,312.123,-71.325,-176.589,7.771,148.502
C08590=1186.370,311.876,-71.294,-176.592,7.768,148.502
C08591=1186.374,311.628,-71.263,-176.594,7.766,148.502
C08592=1186.378,311.380,-71.232,-176.596,7.762,148.502
C08593=1186.383,311.132,-71.202,-176.599,7.759,148.502
C08594=1186.388,310.884,-71.171,-176.602,7.756,148.502
C08595=1186.391,310.635,-71.140,-176.604,7.753,148.501
C08596=1186.395,310.388,-71.109,-176.607,7.750,148.501
C08597=1186.400,310.140,-71.079,-176.609,7.747,148.501
C08598=1186.404,309.891,-71.049,-176.611,7.745,148.501
C08599=1186.408,309.643,-71.018,-176.614,7.741,148.501
C08600=1186.413,309.395,-70.987,-176.616,7.738,148.501
C08601=1186.417,309.147,-70.957,-176.619,7.735,148.501
C08602=1186.421,308.898,-70.926,-176.622,7.732,148.501
C08603=1186.425,308.650,-70.895,-176.624,7.729,148.501
C08604=1186.429,308.403,-70.865,-176.626,7.727,148.501
C08605=1186.434,308.155,-70.834,-176.629,7.724,148.501
C08606=1186.438,307.907,-70.804,-176.632,7.721,148.501
C08607=1186.442,307.658,-70.774,-176.634,7.718,148.501
C08608=1186.447,307.410,-70.743,-176.637,7.715,148.501
C08609=1186.451,307.162,-70.713,-176.639,7.712,148.501
C08610=1186.455,306.914,-70.682,-176.641,7.709,148.501
C08611=1186.458,306.666,-70.652,-176.644,7.706,148.501
C08612=1186.463,306.417,-70.621,-176.646,7.703,148.501
C08613=1186.468,306.169,-70.591,-176.649,7.700,148.501
C08614=1186.472,305.922,-70.561,-176.652,7.697,148.501
C08615=1186.476,305.674,-70.530,-176.654,7.695,148.501
C08616=1186.481,305.426,-70.500,-176.657,7.692,148.501
C08617=1186.485,305.177,-70.469,-176.659,7.689,148.501
C08618=1186.489,304.929,-70.439,-176.662,7.686,148.501
C08619=1186.493,304.681,-70.409,-176.664,7.683,148.501
C08620=1186.497,304.433,-70.379,-176.667,7.680,148.501
C08621=1186.502,304.185,-70.348,-176.669,7.677,148.501
C08622=1186.506,303.937,-70.319,-176.671,7.674,148.501
C08623=1186.510,303.688,-70.287,-176.674,7.671,148.501
C08624=1186.514,303.440,-70.258,-176.677,7.668,148.501
C08625=1186.519,303.192,-70.227,-176.680,7.665,148.501
C08626=1186.523,302.944,-70.197,-176.682,7.663,148.501
C08627=1186.528,302.696,-70.167,-176.684,7.660,148.501
C08628=1186.532,302.448,-70.137,-176.687,7.657,148.501
C08629=1186.536,302.199,-70.107,-176.689,7.654,148.501
C08630=1186.540,301.952,-70.077,-176.692,7.651,148.501
C08631=1186.545,301.704,-70.047,-176.694,7.648,148.501
C08632=1186.549,301.455,-70.016,-176.697,7.645,148.501
C08633=1186.553,301.207,-69.987,-176.700,7.642,148.501
C08634=1186.557,300.959,-69.956,-176.702,7.639,148.501
C08635=1186.562,300.710,-69.926,-176.705,7.636,148.501
C08636=1186.565,300.463,-69.896,-176.707,7.634,148.501
C08637=1186.570,300.214,-69.866,-176.710,7.631,148.501
C08638=1186.574,299.967,-69.836,-176.712,7.628,148.501
C08639=1186.578,299.718,-69.807,-176.715,7.625,148.501
C08640=1186.583,299.470,-69.777,-176.718,7.622,148.501
C08641=1186.587,299.222,-69.746,-176.719,7.620,148.501
C08642=1186.591,298.974,-69.717,-176.722,7.617,148.501
C08643=1186.596,298.726,-69.686,-176.725,7.614,148.501
C08644=1186.600,298.478,-69.657,-176.728,7.611,148.501
C08645=1186.604,298.229,-69.627,-176.730,7.608,148.501
C08646=1186.609,297.981,-69.596,-176.732,7.605,148.501
C08647=1186.613,297.733,-69.567,-176.735,7.602,148.501
C08648=1186.617,297.485,-69.538,-176.738,7.599,148.501
C08649=1186.621,297.237,-69.508,-176.741,7.596,148.501
C08650=1186.626,296.988,-69.477,-176.742,7.594,148.501
C08651=1186.630,296.740,-69.448,-176.745,7.591,148.501
C08652=1186.634,296.491,-69.418,-176.748,7.588,148.501
C08653=1186.638,296.244,-69.388,-176.750,7.585,148.501
C08654=1186.642,295.995,-69.358,-176.753,7.582,148.501
C08655=1186.647,295.747,-69.328,-176.755,7.580,148.501
C08656=1186.651,295.499,-69.299,-176.758,7.577,148.501
C08657=1186.656,295.251,-69.270,-176.761,7.574,148.501
C08658=1186.660,295.003,-69.240,-176.763,7.571,148.501
C08659=1186.664,294.755,-69.210,-176.766,7.569,148.501
C08660=1186.669,294.507,-69.180,-176.768,7.566,148.501
C08661=1186.673,294.258,-69.151,-176.771,7.562,148.501
C08662=1186.677,294.010,-69.121,-176.773,7.559,148.501
C08663=1186.681,293.762,-69.092,-176.775,7.557,148.501
C08664=1186.686,293.513,-69.062,-176.778,7.554,148.501
C08665=1186.690,293.265,-69.033,-176.781,7.551,148.501
C08666=1186.694,293.017,-69.003,-176.784,7.548,148.501
C08667=1186.698,292.769,-68.973,-176.786,7.546,148.501
C08668=1186.703,292.521,-68.943,-176.788,7.543,148.501
C08669=1186.707,292.272,-68.914,-176.791,7.540,148.501
C08670=1186.711,292.024,-68.884,-176.794,7.537,148.501
C08671=1186.715,291.776,-68.855,-176.796,7.535,148.501
C08672=1186.719,291.528,-68.825,-176.799,7.532,148.501
C08673=1186.724,291.280,-68.796,-176.801,7.529,148.501
C08674=1186.728,291.032,-68.767,-176.804,7.526,148.501
C08675=1186.733,290.784,-68.737,-176.806,7.524,148.501
C08676=1186.737,290.535,-68.709,-176.809,7.521,148.502
C08677=1186.741,290.286,-68.679,-176.812,7.518,148.502
C08678=1186.745,290.038,-68.650,-176.814,7.515,148.502
C08679=1186.750,289.790,-68.620,-176.817,7.512,148.502
C08680=1186.754,289.542,-68.591,-176.819,7.509,148.502
C08681=1186.759,289.294,-68.562,-176.822,7.506,148.502
C08682=1186.763,289.046,-68.532,-176.825,7.503,148.502
C08683=1186.768,288.770,-68.500,-176.828,7.500,148.502
C08684=1186.772,288.497,-68.467,-176.830,7.497,148.502
C08685=1186.776,288.222,-68.435,-176.833,7.494,148.502
C08686=1186.782,287.947,-68.403,-176.836,7.491,148.502
C08687=1186.786,287.699,-68.374,-176.838,7.488,148.502
C08688=1186.790,287.450,-68.344,-176.841,7.485,148.502
C08689=1186.794,287.202,-68.315,-176.843,7.483,148.502
C08690=1186.800,286.954,-68.286,-176.846,7.480,148.502
C08691=1186.804,286.706,-68.257,-176.849,7.477,148.502
C08692=1186.807,286.458,-68.228,-176.851,7.474,148.502
C08693=1186.811,286.209,-68.199,-176.854,7.472,148.502
C08694=1186.816,285.960,-68.170,-176.856,7.469,148.502
C08695=1186.821,285.713,-68.141,-176.859,7.466,148.502
C08696=1186.825,285.465,-68.111,-176.861,7.464,148.502
C08697=1186.829,285.216,-68.083,-176.864,7.461,148.502
C08698=1186.833,284.967,-68.053,-176.867,7.458,148.502
C08699=1186.838,284.720,-68.024,-176.869,7.455,148.502
C08700=1186.842,284.471,-67.996,-176.871,7.453,148.502
C08701=1186.846,284.223,-67.966,-176.874,7.450,148.502
C08702=1186.850,283.975,-67.937,-176.877,7.447,148.503
C08703=1186.855,283.727,-67.909,-176.879,7.445,148.503
C08704=1186.860,283.478,-67.879,-176.882,7.442,148.503
C08705=1186.863,283.230,-67.851,-176.885,7.439,148.503
C08706=1186.868,282.982,-67.822,-176.887,7.436,148.503
C08707=1186.873,282.733,-67.793,-176.889,7.433,148.503
C08708=1186.877,282.485,-67.764,-176.892,7.430,148.503
C08709=1186.881,282.236,-67.735,-176.895,7.427,148.503
C08710=1186.885,281.989,-67.707,-176.897,7.425,148.503
C08711=1186.890,281.740,-67.678,-176.900,7.423,148.503
C08712=1186.894,281.492,-67.648,-176.903,7.420,148.503
C08713=1186.899,281.244,-67.620,-176.905,7.417,148.503
C08714=1186.903,280.996,-67.591,-176.908,7.414,148.503
C08715=1186.907,280.747,-67.562,-176.910,7.411,148.503
C08716=1186.911,280.498,-67.533,-176.913,7.409,148.503
C08717=1186.916,280.251,-67.505,-176.915,7.406,148.503
C08718=1186.920,280.002,-67.476,-176.918,7.403,148.503
C08719=1186.924,279.753,-67.447,-176.920,7.401,148.504
C08720=1186.929,279.506,-67.419,-176.923,7.398,148.504
C08721=1186.933,279.257,-67.390,-176.926,7.395,148.504
C08722=1186.937,279.008,-67.361,-176.928,7.393,148.504
C08723=1186.942,278.761,-67.333,-176.931,7.390,148.504
C08724=1186.946,278.512,-67.304,-176.933,7.387,148.504
C08725=1186.950,278.263,-67.275,-176.936,7.384,148.504
C08726=1186.955,278.016,-67.247,-176.939,7.382,148.504
C08727=1186.959,277.767,-67.218,-176.941,7.379,148.504
C08728=1186.963,277.519,-67.190,-176.944,7.376,148.504
C08729=1186.968,277.270,-67.161,-176.946,7.374,148.504
C08730=1186.972,277.022,-67.133,-176.949,7.371,148.504
C08731=1186.976,276.774,-67.104,-176.952,7.368,148.504
C08732=1186.981,276.525,-67.075,-176.954,7.366,148.504
C08733=1186.985,276.278,-67.048,-176.957,7.363,148.504
C08734=1186.990,276.029,-67.019,-176.959,7.360,148.505
C08735=1186.993,275.780,-66.991,-176.962,7.358,148.505
C08736=1186.998,275.533,-66.962,-176.965,7.355,148.505
C08737=1187.002,275.284,-66.933,-176.967,7.353,148.505
C08738=1187.007,275.036,-66.905,-176.969,7.350,148.505
C08739=1187.011,274.787,-66.877,-176.972,7.347,148.505
C08740=1187.016,274.539,-66.849,-176.974,7.345,148.505
C08741=1187.019,274.290,-66.820,-176.977,7.342,148.505
C08742=1187.024,274.042,-66.792,-176.980,7.339,148.505
C08743=1187.028,273.794,-66.763,-176.982,7.337,148.505
C08744=1187.033,273.545,-66.734,-176.985,7.334,148.506
C08745=1187.037,273.298,-66.707,-176.988,7.331,148.506
C08746=1187.041,273.049,-66.678,-176.990,7.329,148.506
C08747=1187.046,272.801,-66.650,-176.993,7.326,148.506
C08748=1187.050,272.552,-66.621,-176.995,7.323,148.506
C08749=1187.055,272.304,-66.594,-176.998,7.321,148.506
C08750=1187.059,272.055,-66.565,-177.000,7.318,148.506
C08751=1187.063,271.807,-66.537,-177.003,7.316,148.506
C08752=1187.067,271.559,-66.509,-177.006,7.313,148.506
C08753=1187.072,271.310,-66.481,-177.008,7.310,148.506
C08754=1187.076,271.062,-66.452,-177.011,7.308,148.506
C08755=1187.081,270.814,-66.424,-177.013,7.305,148.506
C08756=1187.085,270.565,-66.397,-177.016,7.302,148.506
C08757=1187.089,270.317,-66.369,-177.019,7.300,148.507
C08758=1187.094,270.068,-66.340,-177.021,7.297,148.507
C08759=1187.098,269.820,-66.312,-177.024,7.295,148.507
C08760=1187.102,269.571,-66.284,-177.026,7.292,148.507
C08761=1187.107,269.323,-66.256,-177.029,7.289,148.507
C08762=1187.111,269.075,-66.228,-177.031,7.287,148.507
C08763=1187.115,268.827,-66.200,-177.034,7.284,148.507
C08764=1187.121,268.578,-66.172,-177.037,7.282,148.507
C08765=1187.124,268.329,-66.144,-177.039,7.279,148.507
C08766=1187.129,268.081,-66.116,-177.042,7.276,148.507
C08767=1187.133,267.833,-66.088,-177.044,7.274,148.508
C08768=1187.138,267.585,-66.060,-177.047,7.271,148.508
C08769=1187.142,267.335,-66.032,-177.050,7.268,148.508
C08770=1187.146,267.088,-66.005,-177.052,7.266,148.508
C08771=1187.151,266.839,-65.976,-177.055,7.263,148.508
C08772=1187.155,266.591,-65.948,-177.057,7.261,148.508
C08773=1187.159,266.342,-65.921,-177.060,7.258,148.508
C08774=1187.163,266.094,-65.893,-177.062,7.256,148.508
C08775=1187.168,265.846,-65.865,-177.065,7.253,148.508
C08776=1187.173,265.597,-65.837,-177.068,7.250,148.508
C08777=1187.177,265.348,-65.809,-177.070,7.248,148.509
C08778=1187.181,265.101,-65.782,-177.073,7.245,148.509
C08779=1187.186,264.852,-65.755,-177.075,7.243,148.509
C08780=1187.190,264.603,-65.726,-177.078,7.240,148.509
C08781=1187.195,264.355,-65.698,-177.081,7.237,148.509
C08782=1187.199,264.107,-65.671,-177.083,7.235,148.509
C08783=1187.203,263.858,-65.643,-177.086,7.232,148.509
C08784=1187.208,263.610,-65.616,-177.088,7.230,148.509
C08785=1187.212,263.362,-65.588,-177.091,7.227,148.509
C08786=1187.217,263.112,-65.560,-177.093,7.225,148.510
C08787=1187.221,262.840,-65.530,-177.096,7.222,148.510
C08788=1187.226,262.567,-65.500,-177.099,7.219,148.510
C08789=1187.231,262.294,-65.469,-177.102,7.216,148.510
C08790=1187.236,262.021,-65.439,-177.105,7.213,148.510
C08791=1187.240,261.773,-65.411,-177.108,7.210,148.510
C08792=1187.245,261.524,-65.384,-177.110,7.208,148.510
C08793=1187.249,261.276,-65.356,-177.113,7.206,148.511
C08794=1187.253,261.027,-65.328,-177.115,7.203,148.511
C08795=1187.258,260.779,-65.301,-177.118,7.200,148.511
C08796=1187.262,260.531,-65.274,-177.120,7.198,148.511
C08797=1187.266,260.282,-65.246,-177.123,7.196,148.511
C08798=1187.271,260.034,-65.218,-177.126,7.193,148.511
C08799=1187.275,259.785,-65.191,-177.128,7.190,148.511
C08800=1187.279,259.537,-65.163,-177.131,7.187,148.511
C08801=1187.284,259.288,-65.136,-177.134,7.186,148.512
C08802=1187.288,259.040,-65.109,-177.136,7.183,148.512
C08803=1187.293,258.792,-65.081,-177.139,7.180,148.512
C08804=1187.297,258.543,-65.054,-177.142,7.178,148.512
C08805=1187.301,258.294,-65.027,-177.144,7.176,148.512
C08806=1187.306,258.046,-64.999,-177.147,7.173,148.512
C08807=1187.311,257.798,-64.972,-177.149,7.171,148.512
C08808=1187.315,257.549,-64.945,-177.152,7.168,148.513
C08809=1187.319,257.300,-64.918,-177.155,7.165,148.513
C08810=1187.324,257.052,-64.890,-177.157,7.163,148.513
C08811=1187.328,256.804,-64.863,-177.160,7.160,148.513
C08812=1187.333,256.555,-64.836,-177.162,7.158,148.513
C08813=1187.338,256.307,-64.809,-177.165,7.155,148.513
C08814=1187.341,256.058,-64.782,-177.167,7.153,148.513
C08815=1187.345,255.810,-64.754,-177.170,7.150,148.513
C08816=1187.350,255.562,-64.727,-177.173,7.148,148.514
C08817=1187.355,255.313,-64.700,-177.175,7.145,148.514
C08818=1187.359,255.065,-64.673,-177.178,7.143,148.514
C08819=1187.363,254.815,-64.645,-177.181,7.140,148.514
C08820=1187.368,254.567,-64.618,-177.183,7.138,148.514
C08821=1187.372,254.319,-64.591,-177.186,7.135,148.514
C08822=1187.376,254.071,-64.564,-177.188,7.133,148.514
C08823=1187.381,253.822,-64.537,-177.191,7.130,148.514
C08824=1187.385,253.574,-64.510,-177.194,7.128,148.515
C08825=1187.390,253.325,-64.483,-177.196,7.125,148.515
C08826=1187.394,253.076,-64.455,-177.198,7.123,148.515
C08827=1187.398,252.828,-64.429,-177.202,7.121,148.515
C08828=1187.403,252.579,-64.402,-177.204,7.118,148.515
C08829=1187.407,252.331,-64.375,-177.206,7.115,148.515
C08830=1187.412,252.083,-64.348,-177.209,7.114,148.516
C08831=1187.417,251.834,-64.321,-177.212,7.111,148.516
C08832=1187.421,251.586,-64.294,-177.214,7.108,148.516
C08833=1187.425,251.337,-64.267,-177.217,7.106,148.516
C08834=1187.430,251.089,-64.240,-177.219,7.104,148.516
C08835=1187.434,250.840,-64.213,-177.222,7.101,148.516
C08836=1187.438,250.591,-64.186,-177.225,7.099,148.517
C08837=1187.443,250.343,-64.159,-177.227,7.096,148.517
C08838=1187.447,250.094,-64.132,-177.230,7.094,148.517
C08839=1187.451,249.846,-64.106,-177.233,7.091,148.517
C08840=1187.456,249.597,-64.079,-177.235,7.089,148.517
C08841=1187.461,249.349,-64.052,-177.238,7.086,148.517
C08842=1187.465,249.100,-64.026,-177.240,7.084,148.517
C08843=1187.469,248.852,-63.999,-177.243,7.081,148.517
C08844=1187.474,248.603,-63.972,-177.246,7.079,148.518
C08845=1187.478,248.355,-63.945,-177.248,7.077,148.518
C08846=1187.483,248.106,-63.919,-177.251,7.074,148.518
C08847=1187.488,247.858,-63.892,-177.253,7.072,148.518
C08848=1187.491,247.610,-63.865,-177.256,7.069,148.518
C08849=1187.496,247.361,-63.838,-177.259,7.067,148.519
C08850=1187.501,247.113,-63.811,-177.261,7.064,148.519
C08851=1187.505,246.864,-63.785,-177.264,7.062,148.519
C08852=1187.510,246.615,-63.758,-177.267,7.060,148.519
C08853=1187.514,246.367,-63.732,-177.269,7.057,148.519
C08854=1187.519,246.118,-63.706,-177.272,7.055,148.519
C08855=1187.523,245.869,-63.679,-177.274,7.053,148.520
C08856=1187.527,245.621,-63.652,-177.276,7.051,148.520
C08857=1187.532,245.373,-63.625,-177.280,7.048,148.520
C08858=1187.536,245.124,-63.599,-177.282,7.046,148.520
C08859=1187.541,244.875,-63.572,-177.285,7.043,148.520
C08860=1187.545,244.627,-63.546,-177.287,7.041,148.520
C08861=1187.550,244.378,-63.519,-177.290,7.038,148.521
C08862=1187.553,244.130,-63.493,-177.293,7.036,148.521
C08863=1187.558,243.881,-63.467,-177.295,7.033,148.521
C08864=1187.562,243.633,-63.440,-177.298,7.031,148.521
C08865=1187.567,243.384,-63.414,-177.300,7.029,148.521
C08866=1187.571,243.135,-63.387,-177.303,7.026,148.522
C08867=1187.576,242.887,-63.360,-177.305,7.024,148.522
C08868=1187.580,242.638,-63.334,-177.309,7.022,148.522
C08869=1187.585,242.390,-63.307,-177.311,7.020,148.522
C08870=1187.589,242.141,-63.282,-177.314,7.017,148.522
C08871=1187.594,241.892,-63.255,-177.316,7.015,148.522
C08872=1187.598,241.644,-63.229,-177.318,7.013,148.523
C08873=1187.603,241.396,-63.202,-177.322,7.010,148.523
C08874=1187.607,241.147,-63.176,-177.324,7.008,148.523
C08875=1187.611,240.899,-63.150,-177.327,7.005,148.523
C08876=1187.616,240.650,-63.124,-177.329,7.003,148.523
C08877=1187.620,240.401,-63.098,-177.332,7.001,148.524
C08878=1187.625,240.152,-63.071,-177.335,6.998,148.524
C08879=1187.629,239.903,-63.045,-177.337,6.996,148.524
C08880=1187.633,239.655,-63.019,-177.340,6.993,148.524
C08881=1187.639,239.407,-62.993,-177.343,6.992,148.524
C08882=1187.643,239.158,-62.967,-177.345,6.989,148.524
C08883=1187.647,238.910,-62.940,-177.348,6.987,148.525
C08884=1187.652,238.661,-62.914,-177.350,6.985,148.525
C08885=1187.656,238.413,-62.888,-177.353,6.982,148.525
C08886=1187.660,238.164,-62.862,-177.355,6.980,148.525
C08887=1187.666,237.915,-62.836,-177.358,6.978,148.525
C08888=1187.670,237.667,-62.810,-177.361,6.975,148.526
C08889=1187.674,237.418,-62.784,-177.363,6.973,148.526
C08890=1187.679,237.169,-62.757,-177.366,6.970,148.526
C08891=1187.683,236.898,-62.728,-177.369,6.968,148.526
C08892=1187.688,236.627,-62.701,-177.372,6.965,148.526
C08893=1187.693,236.355,-62.673,-177.375,6.963,148.527
C08894=1187.698,236.083,-62.643,-177.377,6.961,148.527
C08895=1187.702,235.834,-62.618,-177.380,6.958,148.527
C08896=1187.707,235.586,-62.592,-177.382,6.956,148.527
C08897=1187.712,235.338,-62.567,-177.386,6.953,148.527
C08898=1187.716,235.089,-62.539,-177.388,6.951,148.528
C08899=1187.720,234.840,-62.514,-177.390,6.949,148.528
C08900=1187.725,234.591,-62.488,-177.394,6.946,148.528
C08901=1187.729,234.343,-62.463,-177.396,6.944,148.528
C08902=1187.734,234.095,-62.437,-177.398,6.943,148.529
C08903=1187.739,233.845,-62.410,-177.401,6.940,148.529
C08904=1187.743,233.597,-62.385,-177.404,6.938,148.529
C08905=1187.747,233.349,-62.359,-177.407,6.935,148.529
C08906=1187.752,233.100,-62.333,-177.409,6.933,148.529
C08907=1187.756,232.852,-62.307,-177.411,6.931,148.530
C08908=1187.761,232.602,-62.281,-177.415,6.928,148.530
C08909=1187.766,232.354,-62.255,-177.417,6.926,148.530
C08910=1187.770,232.106,-62.230,-177.419,6.924,148.530
C08911=1187.774,231.857,-62.204,-177.422,6.921,148.530
C08912=1187.778,231.608,-62.178,-177.425,6.919,148.531
C08913=1187.783,231.360,-62.153,-177.427,6.918,148.531
C08914=1187.787,231.111,-62.127,-177.430,6.915,148.531
C08915=1187.792,230.862,-62.101,-177.433,6.913,148.531
C08916=1187.796,230.614,-62.076,-177.435,6.911,148.531
C08917=1187.801,230.365,-62.050,-177.438,6.908,148.532
C08918=1187.806,230.116,-62.024,-177.440,6.906,148.532
C08919=1187.810,229.868,-61.998,-177.443,6.904,148.532
C08920=1187.815,229.619,-61.973,-177.446,6.901,148.532
C08921=1187.819,229.370,-61.948,-177.448,6.899,148.533
C08922=1187.824,229.122,-61.922,-177.451,6.897,148.533
C08923=1187.828,228.873,-61.896,-177.454,6.894,148.533
C08924=1187.832,228.624,-61.871,-177.456,6.893,148.533
C08925=1187.837,228.376,-61.845,-177.459,6.890,148.533
C08926=1187.841,228.127,-61.820,-177.462,6.888,148.534
C08927=1187.846,227.878,-61.794,-177.464,6.886,148.534
C08928=1187.851,227.630,-61.769,-177.467,6.884,148.534
C08929=1187.855,227.381,-61.743,-177.470,6.881,148.534
C08930=1187.859,227.132,-61.718,-177.472,6.879,148.535
C08931=1187.864,226.884,-61.692,-177.475,6.877,148.535
C08932=1187.868,226.635,-61.667,-177.478,6.875,148.535
C08933=1187.873,226.386,-61.642,-177.480,6.872,148.535
C08934=1187.878,226.138,-61.616,-177.483,6.871,148.536
C08935=1187.882,225.889,-61.590,-177.485,6.868,148.536
C08936=1187.887,225.641,-61.565,-177.488,6.866,148.536
C08937=1187.891,225.391,-61.540,-177.491,6.864,148.536
C08938=1187.895,225.144,-61.515,-177.493,6.861,148.536
C08939=1187.900,224.895,-61.489,-177.496,6.859,148.537
C08940=1187.904,224.645,-61.464,-177.498,6.857,148.537
C08941=1187.909,224.397,-61.439,-177.501,6.855,148.537
C08942=1187.913,224.148,-61.413,-177.504,6.853,148.538
C08943=1187.918,223.900,-61.389,-177.506,6.850,148.538
C08944=1187.923,223.651,-61.363,-177.509,6.849,148.538
C08945=1187.927,223.403,-61.337,-177.512,6.846,148.538
C08946=1187.932,223.153,-61.312,-177.514,6.844,148.538
C08947=1187.936,222.906,-61.288,-177.517,6.842,148.539
C08948=1187.941,222.656,-61.263,-177.520,6.839,148.539
C08949=1187.945,222.408,-61.237,-177.522,6.837,148.539
C08950=1187.950,222.159,-61.212,-177.525,6.835,148.539
C08951=1187.954,221.910,-61.186,-177.527,6.833,148.540
C08952=1187.958,221.662,-61.162,-177.530,6.831,148.540
C08953=1187.963,221.413,-61.137,-177.533,6.829,148.540
C08954=1187.968,221.164,-61.111,-177.535,6.827,148.540
C08955=1187.972,220.915,-61.086,-177.538,6.824,148.541
C08956=1187.977,220.667,-61.061,-177.541,6.822,148.541
C08957=1187.981,220.418,-61.036,-177.543,6.820,148.541
C08958=1187.986,220.170,-61.011,-177.546,6.818,148.541
C08959=1187.990,219.920,-60.986,-177.549,6.816,148.542
C08960=1187.995,219.672,-60.961,-177.551,6.813,148.542
C08961=1187.999,219.423,-60.936,-177.554,6.812,148.542
C08962=1188.004,219.174,-60.911,-177.557,6.810,148.542
C08963=1188.009,218.926,-60.886,-177.559,6.807,148.543
C08964=1188.012,218.677,-60.862,-177.562,6.805,148.543
C08965=1188.017,218.429,-60.836,-177.565,6.803,148.543
C08966=1188.022,218.180,-60.811,-177.567,6.800,148.543
C08967=1188.027,217.931,-60.786,-177.570,6.798,148.544
C08968=1188.030,217.682,-60.761,-177.573,6.797,148.544
C08969=1188.036,217.434,-60.737,-177.575,6.794,148.544
C08970=1188.040,217.184,-60.712,-177.578,6.792,148.544
C08971=1188.044,216.936,-60.687,-177.581,6.790,148.545
C08972=1188.049,216.687,-60.662,-177.583,6.788,148.545
C08973=1188.054,216.438,-60.637,-177.586,6.786,148.545
C08974=1188.058,216.190,-60.613,-177.589,6.783,148.545
C08975=1188.062,215.941,-60.587,-177.591,6.782,148.546
C08976=1188.067,215.693,-60.563,-177.594,6.779,148.546
C08977=1188.071,215.443,-60.538,-177.596,6.778,148.546
C08978=1188.076,215.194,-60.514,-177.600,6.775,148.547
C08979=1188.081,214.947,-60.489,-177.602,6.773,148.547
C08980=1188.085,214.697,-60.464,-177.604,6.771,148.547
C08981=1188.089,214.449,-60.440,-177.607,6.769,148.547
C08982=1188.095,214.200,-60.415,-177.610,6.767,148.548
C08983=1188.099,213.951,-60.390,-177.612,6.765,148.548
C08984=1188.103,213.703,-60.365,-177.615,6.763,148.548
C08985=1188.108,213.454,-60.340,-177.618,6.761,148.548
C08986=1188.112,213.205,-60.316,-177.620,6.758,148.549
C08987=1188.117,212.956,-60.291,-177.623,6.756,148.549
C08988=1188.121,212.707,-60.267,-177.626,6.754,148.549
C08989=1188.126,212.459,-60.242,-177.628,6.752,148.550
C08990=1188.131,212.210,-60.218,-177.631,6.750,148.550
C08991=1188.135,211.961,-60.193,-177.634,6.748,148.550
C08992=1188.139,211.713,-60.168,-177.636,6.746,148.550
C08993=1188.144,211.464,-60.144,-177.639,6.744,148.550
C08994=1188.148,211.215,-60.119,-177.641,6.742,148.551
C08995=1188.154,210.944,-60.093,-177.645,6.739,148.551
C08996=1188.159,210.674,-60.067,-177.647,6.738,148.551
C08997=1188.164,210.404,-60.040,-177.650,6.735,148.552
C08998=1188.168,210.133,-60.013,-177.653,6.733,148.552
C08999=1188.173,209.885,-59.989,-177.656,6.730,148.552
C09000=1188.178,209.636,-59.964,-177.658,6.728,148.552
C09001=1188.182,209.387,-59.940,-177.661,6.726,148.553
C09002=1188.186,209.138,-59.915,-177.664,6.725,148.553
C09003=1188.191,208.890,-59.891,-177.666,6.723,148.553
C09004=1188.196,208.641,-59.867,-177.669,6.720,148.554
C09005=1188.200,208.392,-59.842,-177.672,6.718,148.554
C09006=1188.205,208.143,-59.818,-177.674,6.716,148.554
C09007=1188.209,207.894,-59.794,-177.677,6.714,148.555
C09008=1188.214,207.646,-59.770,-177.679,6.712,148.555
C09009=1188.218,207.397,-59.745,-177.683,6.710,148.555
C09010=1188.223,207.148,-59.720,-177.685,6.708,148.555
C09011=1188.228,206.899,-59.696,-177.688,6.706,148.556
C09012=1188.232,206.651,-59.672,-177.690,6.704,148.556
C09013=1188.238,206.402,-59.648,-177.693,6.702,148.556
C09014=1188.241,206.153,-59.624,-177.696,6.700,148.556
C09015=1188.246,205.904,-59.600,-177.699,6.698,148.557
C09016=1188.251,205.655,-59.575,-177.701,6.696,148.557
C09017=1188.255,205.407,-59.551,-177.703,6.694,148.557
C09018=1188.260,205.158,-59.528,-177.706,6.692,148.558
C09019=1188.264,204.909,-59.503,-177.709,6.689,148.558
C09020=1188.269,204.660,-59.479,-177.712,6.688,148.558
C09021=1188.273,204.412,-59.455,-177.714,6.685,148.558
C09022=1188.278,204.163,-59.431,-177.717,6.684,148.559
C09023=1188.283,203.914,-59.407,-177.719,6.682,148.559
C09024=1188.287,203.665,-59.382,-177.722,6.680,148.559
C09025=1188.292,203.416,-59.359,-177.725,6.677,148.560
C09026=1188.296,203.167,-59.335,-177.728,6.675,148.560
C09027=1188.300,202.919,-59.311,-177.730,6.673,148.560
C09028=1188.306,202.670,-59.287,-177.733,6.672,148.561
C09029=1188.310,202.421,-59.263,-177.735,6.670,148.561
C09030=1188.314,202.172,-59.238,-177.738,6.668,148.561
C09031=1188.319,201.923,-59.215,-177.741,6.665,148.561
C09032=1188.323,201.675,-59.191,-177.744,6.663,148.562
C09033=1188.328,201.426,-59.166,-177.746,6.661,148.562
C09034=1188.333,201.177,-59.143,-177.749,6.660,148.562
C09035=1188.337,200.929,-59.119,-177.752,6.658,148.563
C09036=1188.342,200.679,-59.095,-177.754,6.656,148.563
C09037=1188.346,200.431,-59.071,-177.756,6.654,148.563
C09038=1188.351,200.181,-59.047,-177.760,6.651,148.564
C09039=1188.355,199.933,-59.023,-177.762,6.649,148.564
C09040=1188.360,199.684,-58.999,-177.765,6.648,148.564
C09041=1188.365,199.435,-58.975,-177.767,6.646,148.564
C09042=1188.370,199.186,-58.952,-177.770,6.644,148.565
C09043=1188.374,198.938,-58.928,-177.772,6.642,148.565
C09044=1188.379,198.689,-58.905,-177.775,6.640,148.565
C09045=1188.383,198.440,-58.880,-177.778,6.637,148.566
C09046=1188.388,198.191,-58.857,-177.781,6.636,148.566
C09047=1188.392,197.943,-58.833,-177.783,6.634,148.566
C09048=1188.397,197.694,-58.810,-177.786,6.632,148.567
C09049=1188.402,197.445,-58.786,-177.788,6.630,148.567
C09050=1188.406,197.196,-58.762,-177.791,6.628,148.567
C09051=1188.410,196.947,-58.739,-177.794,6.626,148.568
C09052=1188.415,196.698,-58.714,-177.796,6.625,148.568
C09053=1188.420,196.449,-58.690,-177.799,6.622,148.568
C09054=1188.425,196.200,-58.667,-177.802,6.620,148.568
C09055=1188.429,195.951,-58.643,-177.805,6.618,148.569
C09056=1188.434,195.702,-58.620,-177.807,6.616,148.569
C09057=1188.438,195.453,-58.596,-177.810,6.614,148.569
C09058=1188.443,195.205,-58.572,-177.813,6.613,148.570
C09059=1188.447,194.956,-58.549,-177.815,6.610,148.570
C09060=1188.452,194.707,-58.526,-177.817,6.609,148.570
C09061=1188.456,194.459,-58.502,-177.821,6.606,148.571
C09062=1188.460,194.210,-58.479,-177.823,6.604,148.571
C09063=1188.465,193.961,-58.455,-177.826,6.602,148.571
C09064=1188.470,193.712,-58.432,-177.829,6.601,148.572
C09065=1188.475,193.463,-58.409,-177.831,6.599,148.572
C09066=1188.479,193.214,-58.385,-177.834,6.597,148.572
C09067=1188.484,192.965,-58.361,-177.836,6.595,148.572
C09068=1188.489,192.717,-58.338,-177.839,6.593,148.573
C09069=1188.494,192.468,-58.315,-177.841,6.591,148.573
C09070=1188.498,192.219,-58.291,-177.844,6.589,148.573
C09071=1188.503,191.970,-58.267,-177.847,6.588,148.574
C09072=1188.507,191.721,-58.244,-177.850,6.585,148.574
C09073=1188.512,191.472,-58.221,-177.853,6.583,148.574
C09074=1188.516,191.224,-58.198,-177.855,6.581,148.575
C09075=1188.521,190.975,-58.175,-177.858,6.579,148.575
C09076=1188.526,190.726,-58.151,-177.860,6.578,148.575
C09077=1188.530,190.477,-58.128,-177.863,6.576,148.576
C09078=1188.535,190.227,-58.105,-177.866,6.574,148.576
C09079=1188.540,189.978,-58.081,-177.868,6.572,148.576
C09080=1188.543,189.730,-58.058,-177.871,6.570,148.577
C09081=1188.548,189.481,-58.034,-177.874,6.569,148.577
C09082=1188.553,189.233,-58.011,-177.876,6.567,148.577
C09083=1188.558,188.984,-57.988,-177.878,6.565,148.578
C09084=1188.563,188.735,-57.965,-177.881,6.563,148.578
C09085=1188.567,188.486,-57.941,-177.884,6.560,148.578
C09086=1188.571,188.237,-57.918,-177.887,6.558,148.579
C09087=1188.576,187.988,-57.895,-177.890,6.557,148.579
C09088=1188.581,187.739,-57.872,-177.892,6.555,148.579
C09089=1188.585,187.490,-57.848,-177.895,6.553,148.580
C09090=1188.590,187.242,-57.826,-177.898,6.551,148.580
C09091=1188.595,186.992,-57.803,-177.900,6.549,148.580
C09092=1188.600,186.743,-57.780,-177.903,6.548,148.581
C09093=1188.604,186.494,-57.757,-177.906,6.546,148.581
C09094=1188.608,186.246,-57.734,-177.908,6.544,148.581
C09095=1188.613,185.997,-57.711,-177.910,6.542,148.582
C09096=1188.618,185.748,-57.688,-177.913,6.540,148.582
C09097=1188.622,185.500,-57.665,-177.916,6.538,148.582
C09098=1188.627,185.250,-57.641,-177.918,6.537,148.583
C09099=1188.632,184.981,-57.616,-177.922,6.534,148.583
C09100=1188.637,184.711,-57.592,-177.924,6.532,148.583
C09101=1188.642,184.442,-57.567,-177.927,6.530,148.584
C09102=1188.648,184.172,-57.542,-177.930,6.529,148.584
C09103=1188.652,183.923,-57.519,-177.932,6.527,148.584
C09104=1188.656,183.674,-57.496,-177.936,6.524,148.585
C09105=1188.661,183.425,-57.474,-177.938,6.522,148.585
C09106=1188.666,183.176,-57.451,-177.941,6.521,148.585
C09107=1188.671,182.927,-57.427,-177.944,6.519,148.586
C09108=1188.674,182.679,-57.405,-177.946,6.517,148.586
C09109=1188.679,182.429,-57.382,-177.949,6.515,148.586
C09110=1188.684,182.181,-57.360,-177.952,6.513,148.587
C09111=1188.689,181.932,-57.336,-177.954,6.512,148.587
C09112=1188.693,181.683,-57.313,-177.957,6.510,148.588
C09113=1188.698,181.433,-57.291,-177.960,6.508,148.588
C09114=1188.703,181.185,-57.268,-177.962,6.506,148.588
C09115=1188.707,180.936,-57.245,-177.965,6.504,148.589
C09116=1188.712,180.687,-57.222,-177.968,6.503,148.589
C09117=1188.716,180.438,-57.200,-177.970,6.501,148.589
C09118=1188.721,180.190,-57.177,-177.973,6.499,148.590
C09119=1188.725,179.940,-57.155,-177.976,6.497,148.590
C09120=1188.730,179.691,-57.131,-177.978,6.496,148.590
C09121=1188.734,179.442,-57.109,-177.981,6.493,148.591
C09122=1188.740,179.194,-57.086,-177.983,6.492,148.591
C09123=1188.744,178.945,-57.063,-177.986,6.490,148.591
C09124=1188.749,178.695,-57.041,-177.989,6.488,148.592
C09125=1188.753,178.447,-57.018,-177.991,6.486,148.592
C09126=1188.758,178.198,-56.996,-177.994,6.484,148.592
C09127=1188.762,177.949,-56.973,-177.997,6.483,148.593
C09128=1188.768,177.700,-56.951,-177.999,6.481,148.593
C09129=1188.772,177.451,-56.928,-178.002,6.479,148.593
C09130=1188.777,177.202,-56.905,-178.005,6.477,148.594
C09131=1188.781,176.954,-56.883,-178.007,6.475,148.594
C09132=1188.786,176.704,-56.860,-178.010,6.474,148.595
C09133=1188.790,176.455,-56.837,-178.013,6.472,148.595
C09134=1188.795,176.207,-56.816,-178.015,6.470,148.595
C09135=1188.800,175.958,-56.792,-178.018,6.468,148.596
C09136=1188.804,175.708,-56.770,-178.021,6.467,148.596
C09137=1188.810,175.460,-56.747,-178.023,6.465,148.596
C09138=1188.814,175.211,-56.725,-178.026,6.463,148.597
C09139=1188.818,174.961,-56.703,-178.029,6.461,148.597
